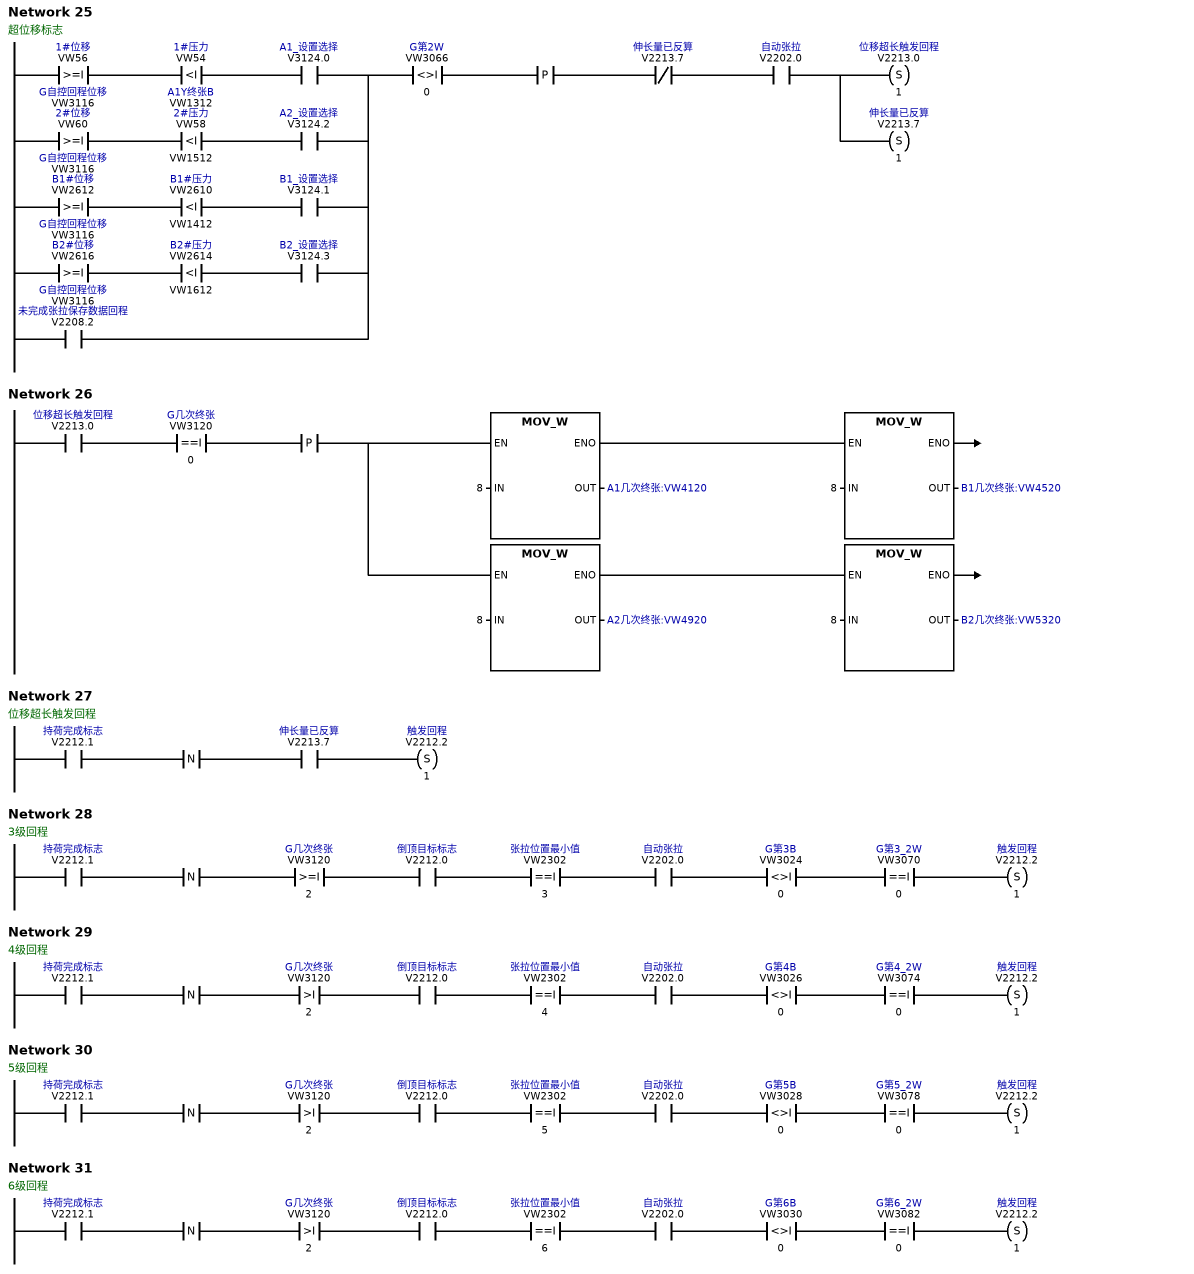
[picture p24: SBR13 networks 25-31]
Network 25
// 超位移标志
LDW>=  1#位移:VW56, G自控回程位移:VW3116
AW<    1#压力:VW54, A1Y终张B:VW1312
A      A1_设置选择:V3124.0
LDW>=  2#位移:VW60, G自控回程位移:VW3116
AW<    2#压力:VW58, VW1512
A      A2_设置选择:V3124.2
OLD
LDW>=  B1#位移:VW2612, G自控回程位移:VW3116
AW<    B1#压力:VW2610, VW1412
A      B1_设置选择:V3124.1
OLD
LDW>=  B2#位移:VW2616, G自控回程位移:VW3116
AW<    B2#压力:VW2614, VW1612
A      B2_设置选择:V3124.3
OLD
O      未完成张拉保存数据回程:V2208.2
AW<>   G第2W:VW3066, 0
EU
AN     伸长量已反算:V2213.7
A      自动张拉:V2202.0
S      位移超长触发回程:V2213.0, 1
S      伸长量已反算:V2213.7, 1
Network 26
LD     位移超长触发回程:V2213.0
AW=    G几次终张:VW3120, 0
EU
LPS
MOVW   8, A1几次终张:VW4120
AENO
MOVW   8, B1几次终张:VW4520
LPP
MOVW   8, A2几次终张:VW4920
AENO
MOVW   8, B2几次终张:VW5320
Network 27
// 位移超长触发回程
LD     持荷完成标志:V2212.1
ED
A      伸长量已反算:V2213.7
S      触发回程:V2212.2, 1
Network 28
// 3级回程
LD     持荷完成标志:V2212.1
ED
AW>=   G几次终张:VW3120, 2
A      倒顶目标标志:V2212.0
AW=    张拉位置最小值:VW2302, 3
A      自动张拉:V2202.0
AW<>   G第3B:VW3024, 0
AW=    G第3_2W:VW3070, 0
S      触发回程:V2212.2, 1
Network 29
// 4级回程
LD     持荷完成标志:V2212.1
ED
AW>    G几次终张:VW3120, 2
A      倒顶目标标志:V2212.0
AW=    张拉位置最小值:VW2302, 4
A      自动张拉:V2202.0
AW<>   G第4B:VW3026, 0
AW=    G第4_2W:VW3074, 0
S      触发回程:V2212.2, 1
Network 30
// 5级回程
LD     持荷完成标志:V2212.1
ED
AW>    G几次终张:VW3120, 2
A      倒顶目标标志:V2212.0
AW=    张拉位置最小值:VW2302, 5
A      自动张拉:V2202.0
AW<>   G第5B:VW3028, 0
AW=    G第5_2W:VW3078, 0
S      触发回程:V2212.2, 1
Network 31
// 6级回程
LD     持荷完成标志:V2212.1
ED
AW>    G几次终张:VW3120, 2
A      倒顶目标标志:V2212.0
AW=    张拉位置最小值:VW2302, 6
A      自动张拉:V2202.0
AW<>   G第6B:VW3030, 0
AW=    G第6_2W:VW3082, 0
S      触发回程:V2212.2, 1
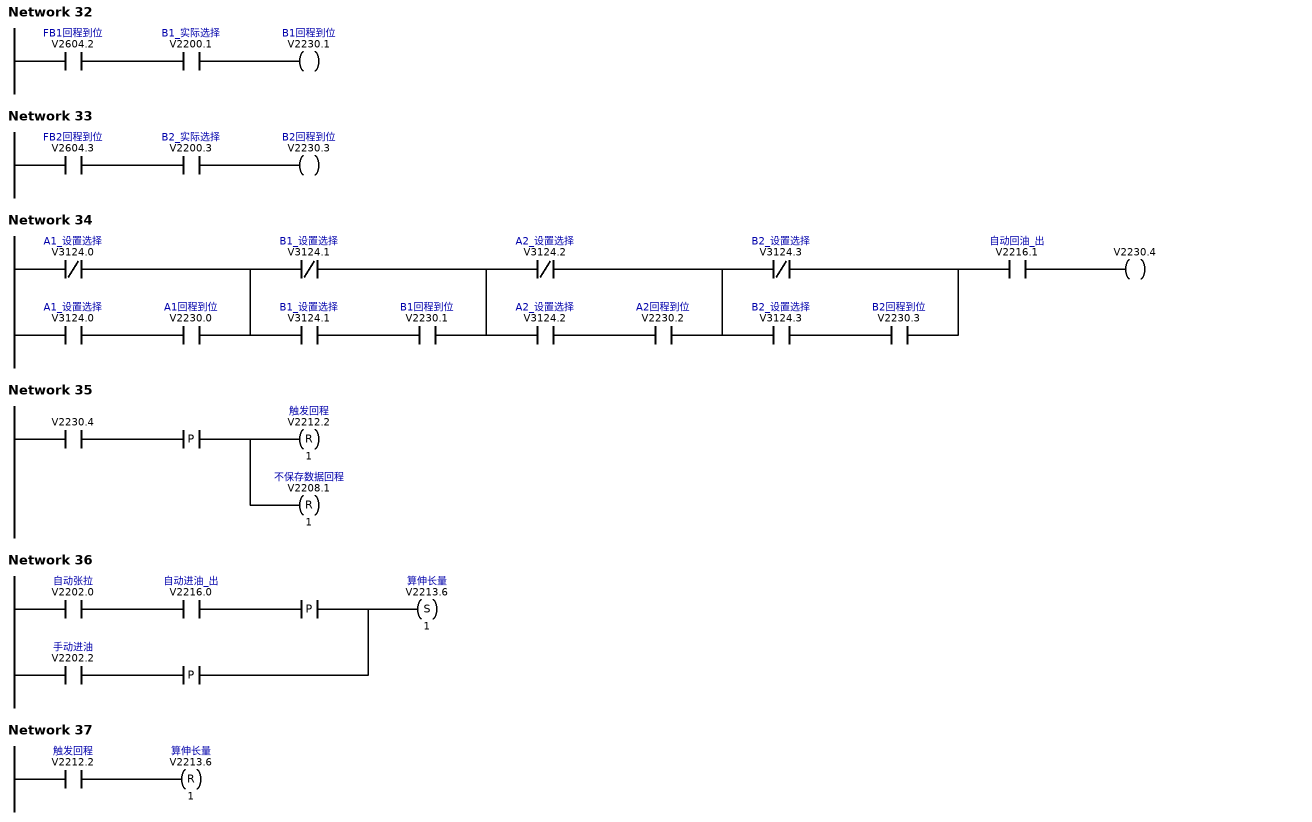
Network 32
LD     FB1回程到位:V2604.2
A      B1_实际选择:V2200.1
=      B1回程到位:V2230.1
Network 33
LD     FB2回程到位:V2604.3
A      B2_实际选择:V2200.3
=      B2回程到位:V2230.3
Network 34
LDN    A1_设置选择:V3124.0
LD     A1_设置选择:V3124.0
A      A1回程到位:V2230.0
OLD
LDN    B1_设置选择:V3124.1
LD     B1_设置选择:V3124.1
A      B1回程到位:V2230.1
OLD
ALD
LDN    A2_设置选择:V3124.2
LD     A2_设置选择:V3124.2
A      A2回程到位:V2230.2
OLD
ALD
LDN    B2_设置选择:V3124.3
LD     B2_设置选择:V3124.3
A      B2回程到位:V2230.3
OLD
ALD
A      自动回油_出:V2216.1
=      V2230.4
Network 35
LD     V2230.4
EU
R      触发回程:V2212.2, 1
R      不保存数据回程:V2208.1, 1
Network 36
LD     自动张拉:V2202.0
A      自动进油_出:V2216.0
EU
LD     手动进油:V2202.2
EU
OLD
S      算伸长量:V2213.6, 1
Network 37
LD     触发回程:V2212.2
R      算伸长量:V2213.6, 1
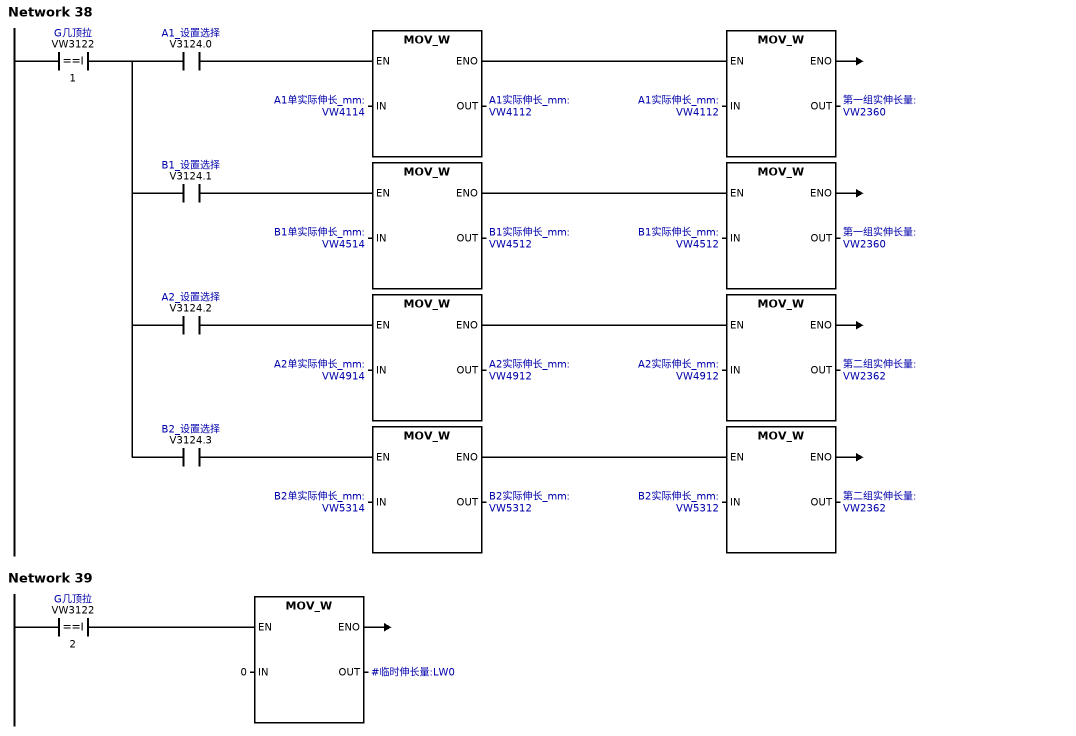
Network 38
LDW=   G几顶拉:VW3122, 1
LPS
A      A1_设置选择:V3124.0
MOVW   A1单实际伸长_mm:VW4114, A1实际伸长_mm:VW4112
AENO
MOVW   A1实际伸长_mm:VW4112, 第一组实伸长量:VW2360
LRD
A      B1_设置选择:V3124.1
MOVW   B1单实际伸长_mm:VW4514, B1实际伸长_mm:VW4512
AENO
MOVW   B1实际伸长_mm:VW4512, 第一组实伸长量:VW2360
LRD
A      A2_设置选择:V3124.2
MOVW   A2单实际伸长_mm:VW4914, A2实际伸长_mm:VW4912
AENO
MOVW   A2实际伸长_mm:VW4912, 第二组实伸长量:VW2362
LPP
A      B2_设置选择:V3124.3
MOVW   B2单实际伸长_mm:VW5314, B2实际伸长_mm:VW5312
AENO
MOVW   B2实际伸长_mm:VW5312, 第二组实伸长量:VW2362
Network 39
LDW=   G几顶拉:VW3122, 2
MOVW   0, #临时伸长量:LW0
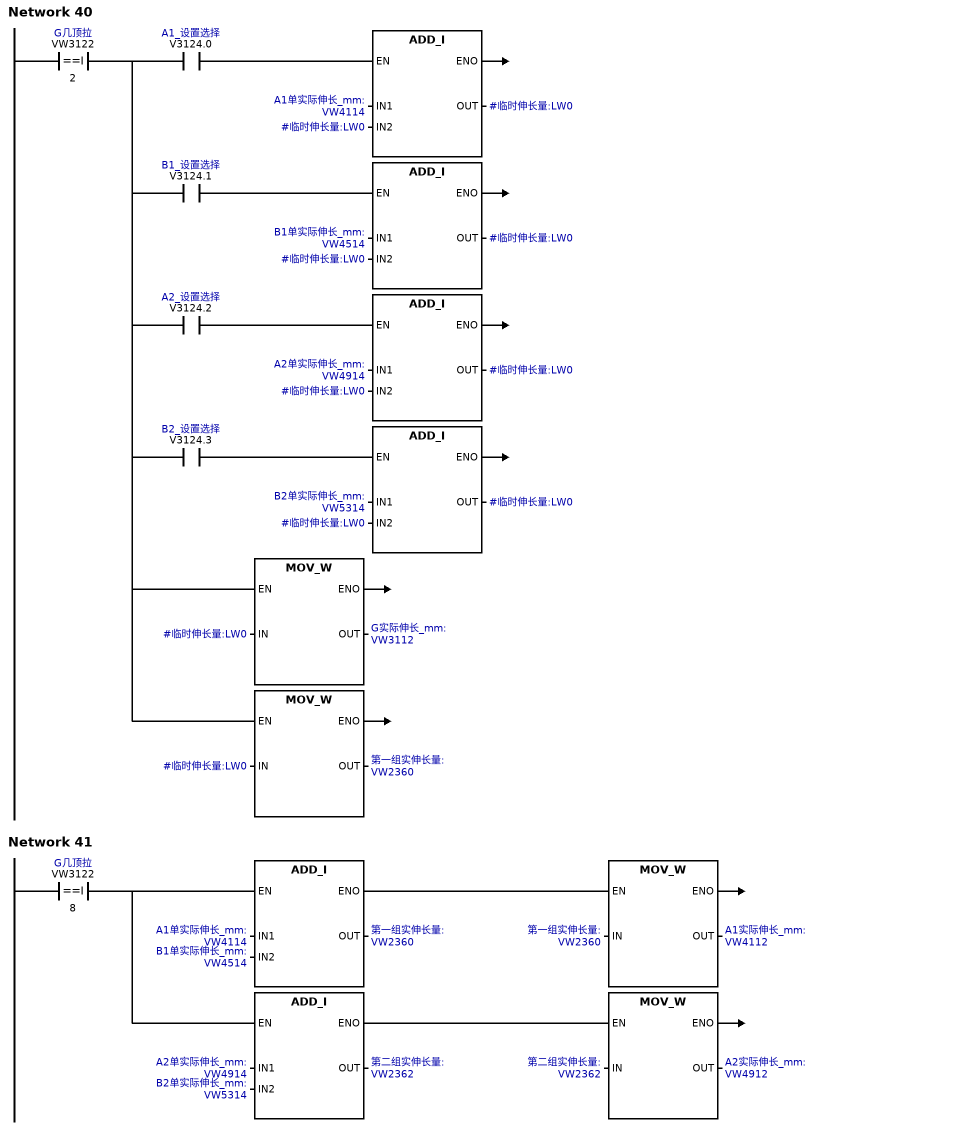
Network 40
LDW=   G几顶拉:VW3122, 2
LPS
A      A1_设置选择:V3124.0
+I     A1单实际伸长_mm:VW4114, #临时伸长量:LW0
LRD
A      B1_设置选择:V3124.1
+I     B1单实际伸长_mm:VW4514, #临时伸长量:LW0
LRD
A      A2_设置选择:V3124.2
+I     A2单实际伸长_mm:VW4914, #临时伸长量:LW0
LRD
A      B2_设置选择:V3124.3
+I     B2单实际伸长_mm:VW5314, #临时伸长量:LW0
LRD
MOVW   #临时伸长量:LW0, G实际伸长_mm:VW3112
LPP
MOVW   #临时伸长量:LW0, 第一组实伸长量:VW2360
Network 41
LDW=   G几顶拉:VW3122, 8
LPS
MOVW   A1单实际伸长_mm:VW4114, 第一组实伸长量:VW2360
AENO
+I     B1单实际伸长_mm:VW4514, 第一组实伸长量:VW2360
AENO
MOVW   第一组实伸长量:VW2360, A1实际伸长_mm:VW4112
LPP
MOVW   A2单实际伸长_mm:VW4914, 第二组实伸长量:VW2362
AENO
+I     B2单实际伸长_mm:VW5314, 第二组实伸长量:VW2362
AENO
MOVW   第二组实伸长量:VW2362, A2实际伸长_mm:VW4912
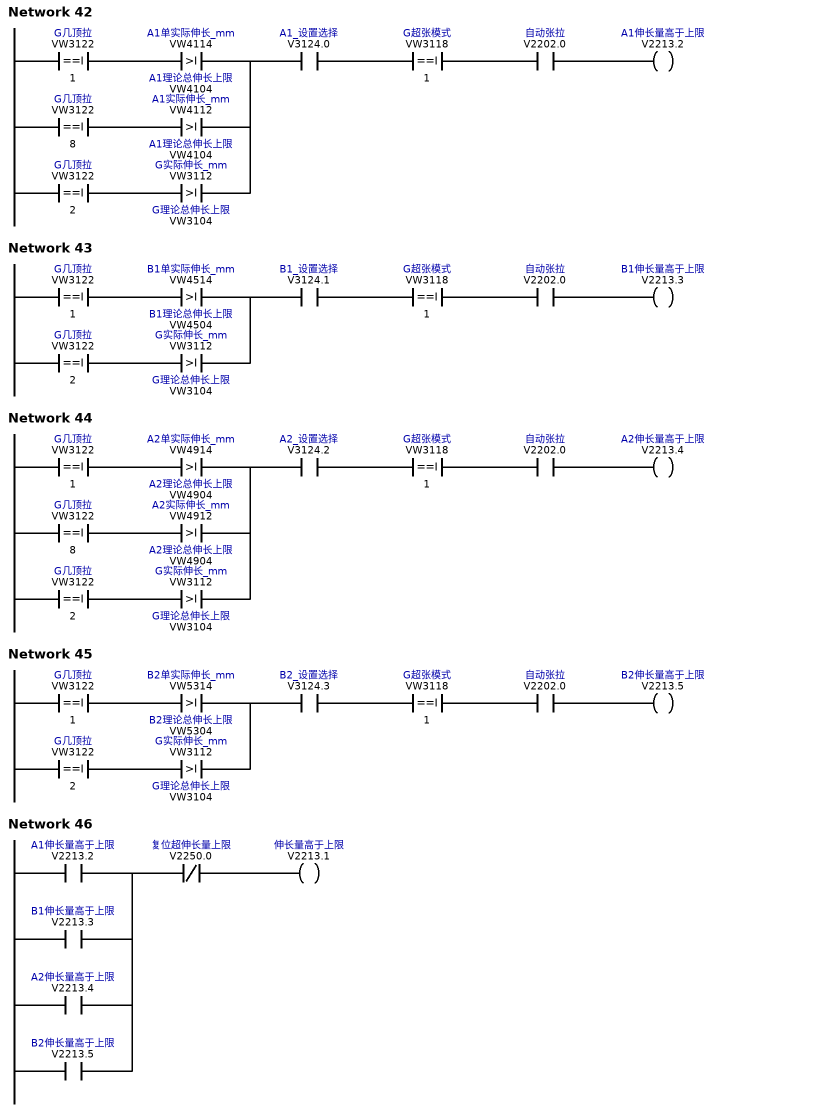
Network 42
LDW=   G几顶拉:VW3122, 1
AW>    A1单实际伸长_mm:VW4114, A1理论总伸长上限:VW4104
LDW=   G几顶拉:VW3122, 8
AW>    A1实际伸长_mm:VW4112, A1理论总伸长上限:VW4104
OLD
LDW=   G几顶拉:VW3122, 2
AW>    G实际伸长_mm:VW3112, G理论总伸长上限:VW3104
OLD
A      A1_设置选择:V3124.0
AW=    G超张模式:VW3118, 1
A      自动张拉:V2202.0
=      A1伸长量高于上限:V2213.2
Network 43
LDW=   G几顶拉:VW3122, 1
AW>    B1单实际伸长_mm:VW4514, B1理论总伸长上限:VW4504
LDW=   G几顶拉:VW3122, 2
AW>    G实际伸长_mm:VW3112, G理论总伸长上限:VW3104
OLD
A      B1_设置选择:V3124.1
AW=    G超张模式:VW3118, 1
A      自动张拉:V2202.0
=      B1伸长量高于上限:V2213.3
Network 44
LDW=   G几顶拉:VW3122, 1
AW>    A2单实际伸长_mm:VW4914, A2理论总伸长上限:VW4904
LDW=   G几顶拉:VW3122, 8
AW>    A2实际伸长_mm:VW4912, A2理论总伸长上限:VW4904
OLD
LDW=   G几顶拉:VW3122, 2
AW>    G实际伸长_mm:VW3112, G理论总伸长上限:VW3104
OLD
A      A2_设置选择:V3124.2
AW=    G超张模式:VW3118, 1
A      自动张拉:V2202.0
=      A2伸长量高于上限:V2213.4
Network 45
LDW=   G几顶拉:VW3122, 1
AW>    B2单实际伸长_mm:VW5314, B2理论总伸长上限:VW5304
LDW=   G几顶拉:VW3122, 2
AW>    G实际伸长_mm:VW3112, G理论总伸长上限:VW3104
OLD
A      B2_设置选择:V3124.3
AW=    G超张模式:VW3118, 1
A      自动张拉:V2202.0
=      B2伸长量高于上限:V2213.5
Network 46
LD     A1伸长量高于上限:V2213.2
O      B1伸长量高于上限:V2213.3
O      A2伸长量高于上限:V2213.4
O      B2伸长量高于上限:V2213.5
AN     复位超伸长量上限:V2250.0
=      伸长量高于上限:V2213.1
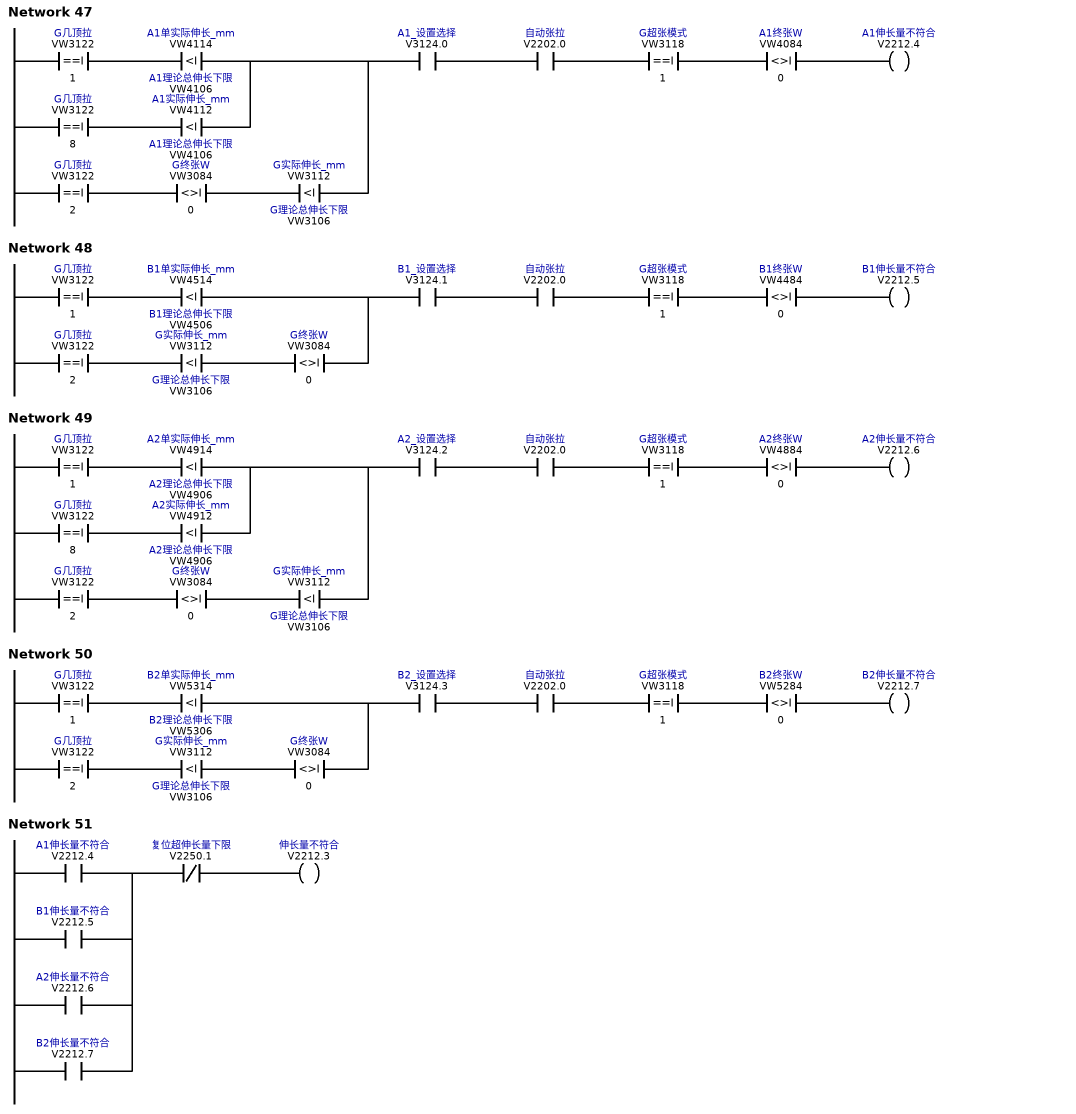
Network 47
LDW=   G几顶拉:VW3122, 1
AW<    A1单实际伸长_mm:VW4114, A1理论总伸长下限:VW4106
LDW=   G几顶拉:VW3122, 8
AW<    A1实际伸长_mm:VW4112, A1理论总伸长下限:VW4106
OLD
LDW=   G几顶拉:VW3122, 2
AW<>   G终张W:VW3084, 0
AW<    G实际伸长_mm:VW3112, G理论总伸长下限:VW3106
OLD
A      A1_设置选择:V3124.0
A      自动张拉:V2202.0
AW=    G超张模式:VW3118, 1
AW<>   A1终张W:VW4084, 0
=      A1伸长量不符合:V2212.4
Network 48
LDW=   G几顶拉:VW3122, 1
AW<    B1单实际伸长_mm:VW4514, B1理论总伸长下限:VW4506
LDW=   G几顶拉:VW3122, 2
AW<    G实际伸长_mm:VW3112, G理论总伸长下限:VW3106
AW<>   G终张W:VW3084, 0
OLD
A      B1_设置选择:V3124.1
A      自动张拉:V2202.0
AW=    G超张模式:VW3118, 1
AW<>   B1终张W:VW4484, 0
=      B1伸长量不符合:V2212.5
Network 49
LDW=   G几顶拉:VW3122, 1
AW<    A2单实际伸长_mm:VW4914, A2理论总伸长下限:VW4906
LDW=   G几顶拉:VW3122, 8
AW<    A2实际伸长_mm:VW4912, A2理论总伸长下限:VW4906
OLD
LDW=   G几顶拉:VW3122, 2
AW<>   G终张W:VW3084, 0
AW<    G实际伸长_mm:VW3112, G理论总伸长下限:VW3106
OLD
A      A2_设置选择:V3124.2
A      自动张拉:V2202.0
AW=    G超张模式:VW3118, 1
AW<>   A2终张W:VW4884, 0
=      A2伸长量不符合:V2212.6
Network 50
LDW=   G几顶拉:VW3122, 1
AW<    B2单实际伸长_mm:VW5314, B2理论总伸长下限:VW5306
LDW=   G几顶拉:VW3122, 2
AW<    G实际伸长_mm:VW3112, G理论总伸长下限:VW3106
AW<>   G终张W:VW3084, 0
OLD
A      B2_设置选择:V3124.3
A      自动张拉:V2202.0
AW=    G超张模式:VW3118, 1
AW<>   B2终张W:VW5284, 0
=      B2伸长量不符合:V2212.7
Network 51
LD     A1伸长量不符合:V2212.4
O      B1伸长量不符合:V2212.5
O      A2伸长量不符合:V2212.6
O      B2伸长量不符合:V2212.7
AN     复位超伸长量下限:V2250.1
=      伸长量不符合:V2212.3
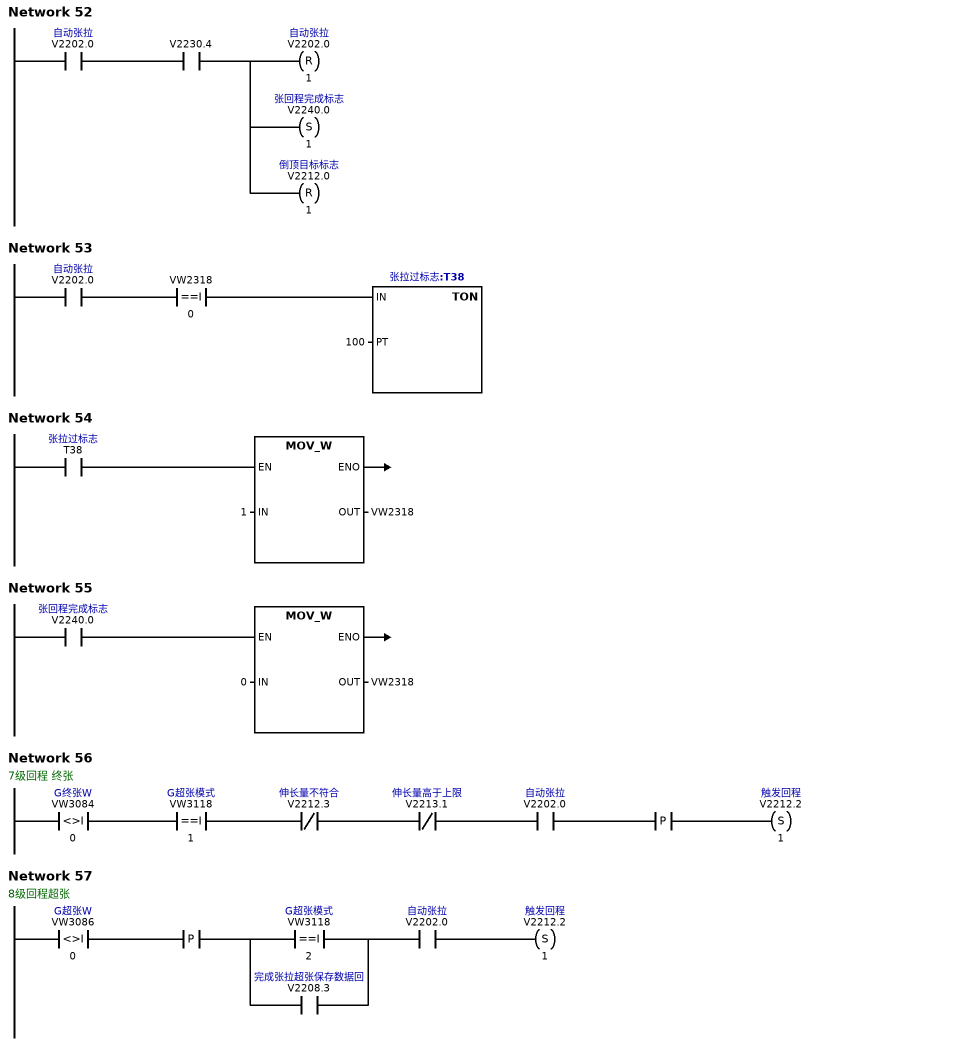
Network 52
LD     自动张拉:V2202.0
A      V2230.4
R      自动张拉:V2202.0, 1
S      张回程完成标志:V2240.0, 1
R      倒顶目标标志:V2212.0, 1
Network 53
LD     自动张拉:V2202.0
AW=    VW2318, 0
TON    张拉过标志:T38, 100
Network 54
LD     张拉过标志:T38
MOVW   1, VW2318
Network 55
LD     张回程完成标志:V2240.0
MOVW   0, VW2318
Network 56
// 7级回程 终张
LDW<>  G终张W:VW3084, 0
AW=    G超张模式:VW3118, 1
AN     伸长量不符合:V2212.3
AN     伸长量高于上限:V2213.1
A      自动张拉:V2202.0
EU
S      触发回程:V2212.2, 1
Network 57
// 8级回程超张
LDW<>  G超张W:VW3086, 0
EU
LDW=   G超张模式:VW3118, 2
O      完成张拉超张保存数据回:V2208.3
ALD
A      自动张拉:V2202.0
S      触发回程:V2212.2, 1
END_SUBROUTINE_BLOCK

SUBROUTINE_BLOCK 自动控制标志:SBR14
TITLE=子程序注释
BEGIN
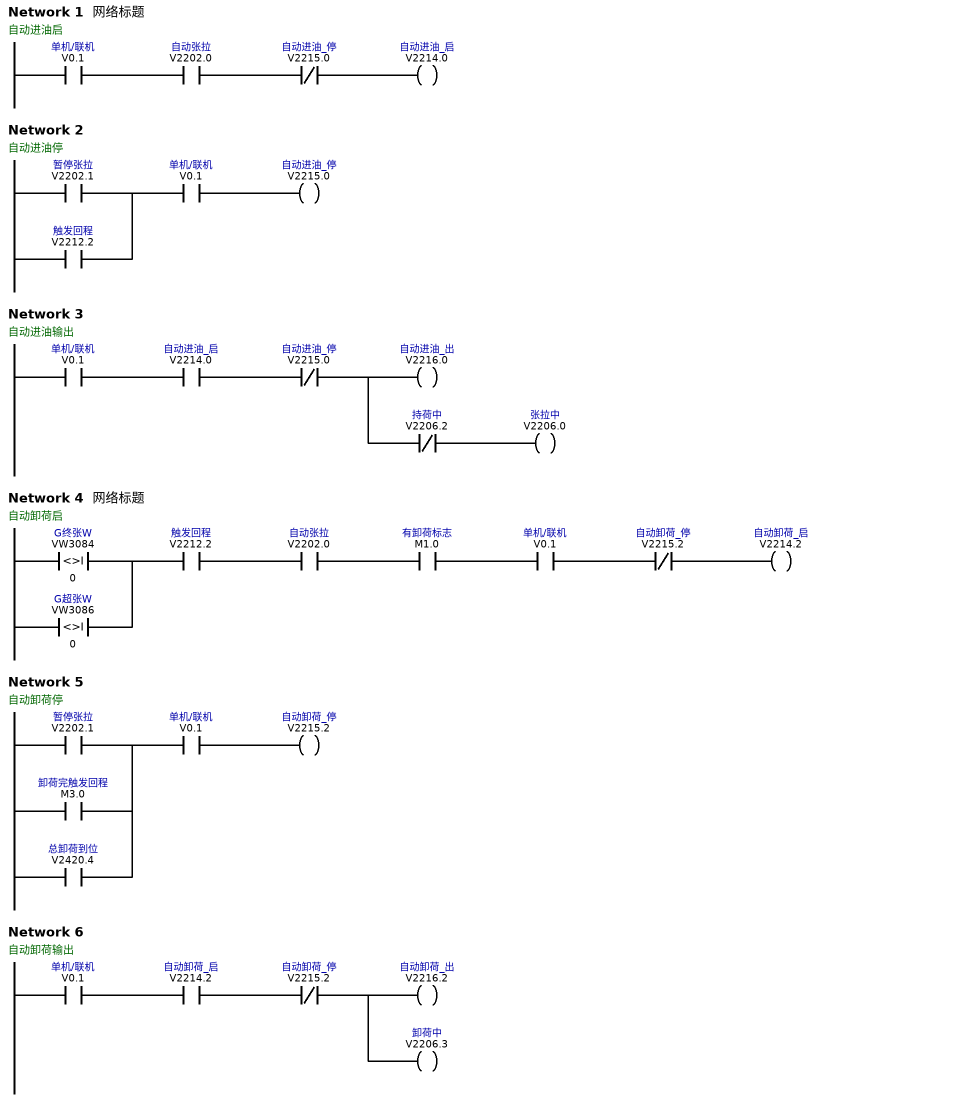
Network 1 // 网络标题
// 自动进油启
LD     单机/联机:V0.1
A      自动张拉:V2202.0
AN     自动进油_停:V2215.0
=      自动进油_启:V2214.0
Network 2
// 自动进油停
LD     暂停张拉:V2202.1
O      触发回程:V2212.2
A      单机/联机:V0.1
=      自动进油_停:V2215.0
Network 3
// 自动进油输出
LD     单机/联机:V0.1
A      自动进油_启:V2214.0
AN     自动进油_停:V2215.0
=      自动进油_出:V2216.0
AN     持荷中:V2206.2
=      张拉中:V2206.0
Network 4 // 网络标题
// 自动卸荷启
LDW<>  G终张W:VW3084, 0
OW<>   G超张W:VW3086, 0
A      触发回程:V2212.2
A      自动张拉:V2202.0
A      有卸荷标志:M1.0
A      单机/联机:V0.1
AN     自动卸荷_停:V2215.2
=      自动卸荷_启:V2214.2
Network 5
// 自动卸荷停
LD     暂停张拉:V2202.1
O      卸荷完触发回程:M3.0
O      总卸荷到位:V2420.4
A      单机/联机:V0.1
=      自动卸荷_停:V2215.2
Network 6
// 自动卸荷输出
LD     单机/联机:V0.1
A      自动卸荷_启:V2214.2
AN     自动卸荷_停:V2215.2
=      自动卸荷_出:V2216.2
=      卸荷中:V2206.3
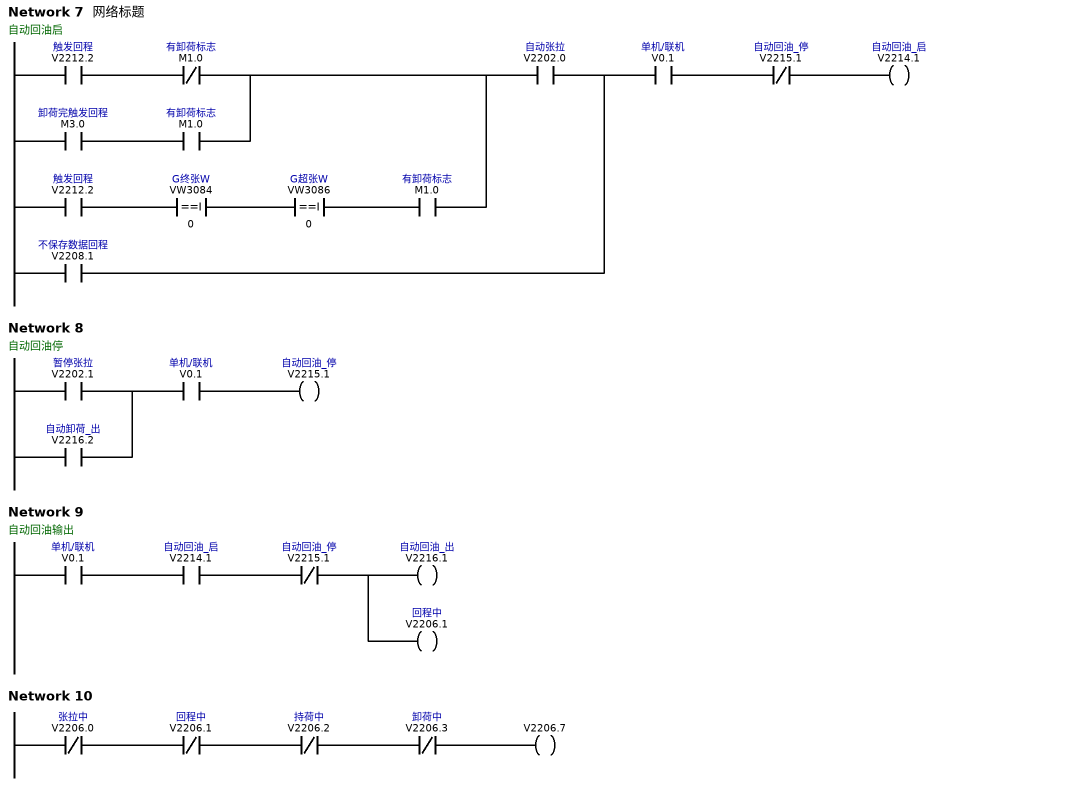
Network 7 // 网络标题
// 自动回油启
LD     触发回程:V2212.2
AN     有卸荷标志:M1.0
LD     卸荷完触发回程:M3.0
A      有卸荷标志:M1.0
OLD
LD     触发回程:V2212.2
AW=    G终张W:VW3084, 0
AW=    G超张W:VW3086, 0
A      有卸荷标志:M1.0
OLD
A      自动张拉:V2202.0
O      不保存数据回程:V2208.1
A      单机/联机:V0.1
AN     自动回油_停:V2215.1
=      自动回油_启:V2214.1
Network 8
// 自动回油停
LD     暂停张拉:V2202.1
O      自动卸荷_出:V2216.2
A      单机/联机:V0.1
=      自动回油_停:V2215.1
Network 9
// 自动回油输出
LD     单机/联机:V0.1
A      自动回油_启:V2214.1
AN     自动回油_停:V2215.1
=      自动回油_出:V2216.1
=      回程中:V2206.1
Network 10
LDN    张拉中:V2206.0
AN     回程中:V2206.1
AN     持荷中:V2206.2
AN     卸荷中:V2206.3
=      V2206.7
END_SUBROUTINE_BLOCK

SUBROUTINE_BLOCK 反算百分比:SBR15
TITLE=子程序注释
VAR_INPUT
当前力:REAL;	// LD0 
总力:REAL;	// LD4 
END_VAR
VAR_OUTPUT
百分比:INT;	// LW8 
END_VAR
VAR
实数百分比:REAL;	// LD10 
END_VAR
BEGIN
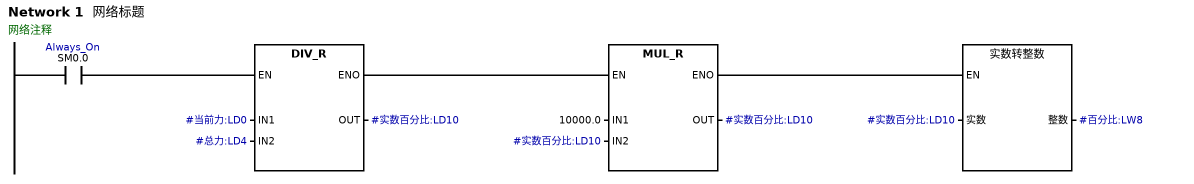
Network 1 // 网络标题
// 网络注释
LD     Always_On:SM0.0
MOVR   #当前力:LD0, #实数百分比:LD10
AENO
/R     #总力:LD4, #实数百分比:LD10
AENO
*R     10000.0, #实数百分比:LD10
AENO
CALL   实数转整数:SBR16, #实数百分比:LD10, #百分比:LW8
END_SUBROUTINE_BLOCK

SUBROUTINE_BLOCK 实数转整数:SBR16
TITLE=子程序注释
VAR_INPUT
实数:REAL;	// LD0 
END_VAR
VAR_OUTPUT
整数:INT;	// LW4 
END_VAR
VAR
双整:DINT;	// LD6 
END_VAR
BEGIN
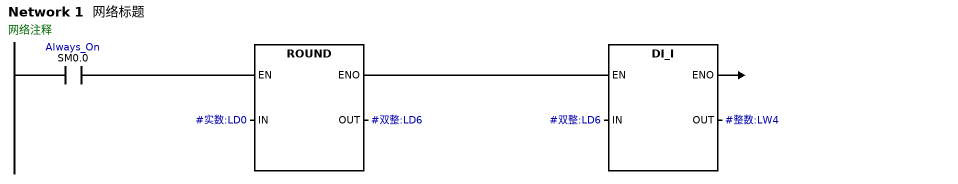
Network 1 // 网络标题
// 网络注释
LD     Always_On:SM0.0
ROUND  #实数:LD0, #双整:LD6
AENO
DTI    #双整:LD6, #整数:LW4
END_SUBROUTINE_BLOCK

SUBROUTINE_BLOCK 计算伸长量:SBR17
TITLE=子程序注释
VAR_INPUT
W1:INT;	// LW0 
W2:INT;	// LW2 
W3_1:INT;	// LW4 
W3_2:INT;	// LW6 
W4_1:INT;	// LW8 
W4_2:INT;	// LW10 
W5_1:INT;	// LW12 
W5_2:INT;	// LW14 
W6_1:INT;	// LW16 
W6_2:INT;	// LW18 
WZZ:INT;	// LW20 
WCZ:INT;	// LW22 
WHS:INT;	// LW24 回缩
当前位移:INT;	// LW26 
WQNSC:INT;	// LW28 千斤顶内伸长量
END_VAR
VAR_OUTPUT
伸长量:INT;	// LW30 
END_VAR
VAR
临时伸长量:INT;	// LW32 
w3差值:INT;	// LW34 
w4差值:INT;	// LW36 
w5差值:INT;	// LW38 
w6差值:INT;	// LW40 
最终值:INT;	// LW42 
初始位移和:INT;	// LW44 
END_VAR
BEGIN
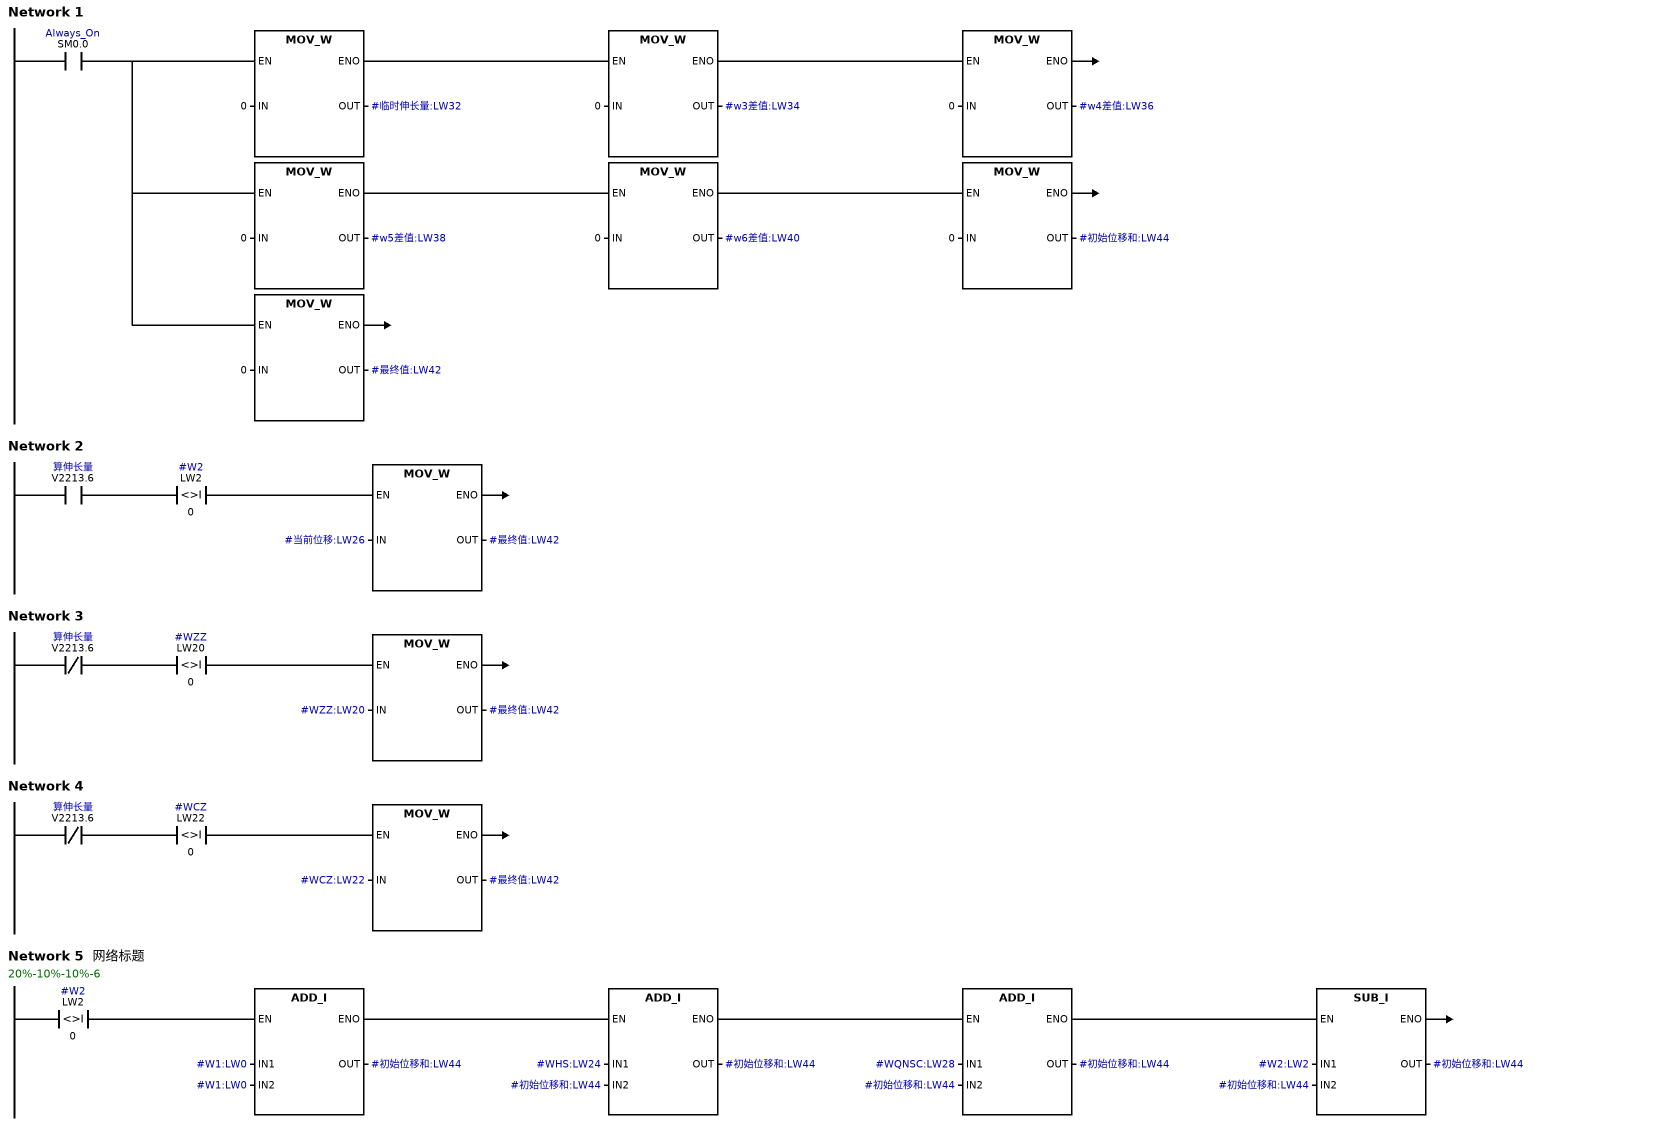
Network 1
LD     Always_On:SM0.0
LPS
MOVW   0, #临时伸长量:LW32
AENO
MOVW   0, #w3差值:LW34
AENO
MOVW   0, #w4差值:LW36
LRD
MOVW   0, #w5差值:LW38
AENO
MOVW   0, #w6差值:LW40
AENO
MOVW   0, #初始位移和:LW44
LPP
MOVW   0, #最终值:LW42
Network 2
LD     算伸长量:V2213.6
AW<>   #W2:LW2, 0
MOVW   #当前位移:LW26, #最终值:LW42
Network 3
LDN    算伸长量:V2213.6
AW<>   #WZZ:LW20, 0
MOVW   #WZZ:LW20, #最终值:LW42
Network 4
LDN    算伸长量:V2213.6
AW<>   #WCZ:LW22, 0
MOVW   #WCZ:LW22, #最终值:LW42
Network 5 // 网络标题
// 20%-10%-10%-6
LDW<>  #W2:LW2, 0
MOVW   #W1:LW0, #初始位移和:LW44
AENO
+I     #W1:LW0, #初始位移和:LW44
AENO
+I     #WHS:LW24, #初始位移和:LW44
AENO
+I     #WQNSC:LW28, #初始位移和:LW44
AENO
INVW   #初始位移和:LW44
INCW   #初始位移和:LW44
+I     #W2:LW2, #初始位移和:LW44
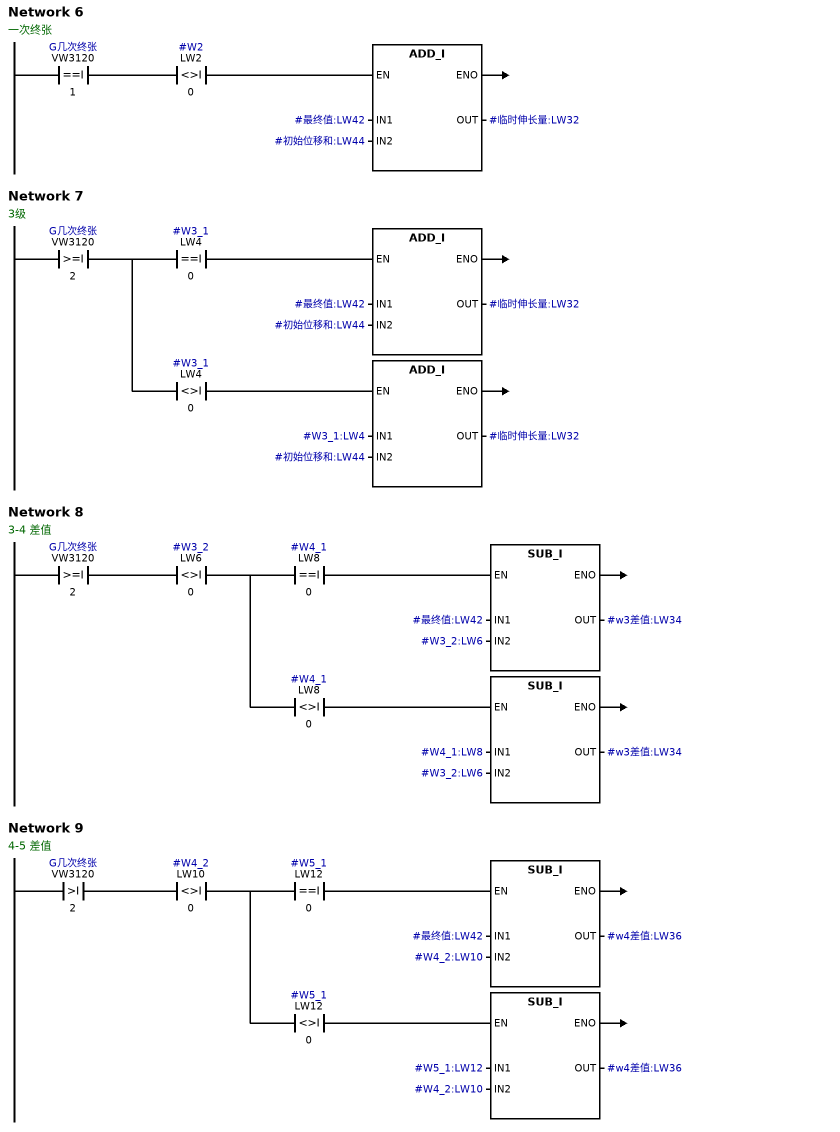
Network 6
// 一次终张
LDW=   G几次终张:VW3120, 1
AW<>   #W2:LW2, 0
MOVW   #最终值:LW42, #临时伸长量:LW32
+I     #初始位移和:LW44, #临时伸长量:LW32
Network 7
// 3级
LDW>=  G几次终张:VW3120, 2
LPS
AW=    #W3_1:LW4, 0
MOVW   #最终值:LW42, #临时伸长量:LW32
+I     #初始位移和:LW44, #临时伸长量:LW32
LPP
AW<>   #W3_1:LW4, 0
MOVW   #W3_1:LW4, #临时伸长量:LW32
+I     #初始位移和:LW44, #临时伸长量:LW32
Network 8
// 3-4 差值
LDW>=  G几次终张:VW3120, 2
AW<>   #W3_2:LW6, 0
LPS
AW=    #W4_1:LW8, 0
MOVW   #最终值:LW42, #w3差值:LW34
-I     #W3_2:LW6, #w3差值:LW34
LPP
AW<>   #W4_1:LW8, 0
MOVW   #W4_1:LW8, #w3差值:LW34
-I     #W3_2:LW6, #w3差值:LW34
Network 9
// 4-5 差值
LDW>   G几次终张:VW3120, 2
AW<>   #W4_2:LW10, 0
LPS
AW=    #W5_1:LW12, 0
MOVW   #最终值:LW42, #w4差值:LW36
-I     #W4_2:LW10, #w4差值:LW36
LPP
AW<>   #W5_1:LW12, 0
MOVW   #W5_1:LW12, #w4差值:LW36
-I     #W4_2:LW10, #w4差值:LW36
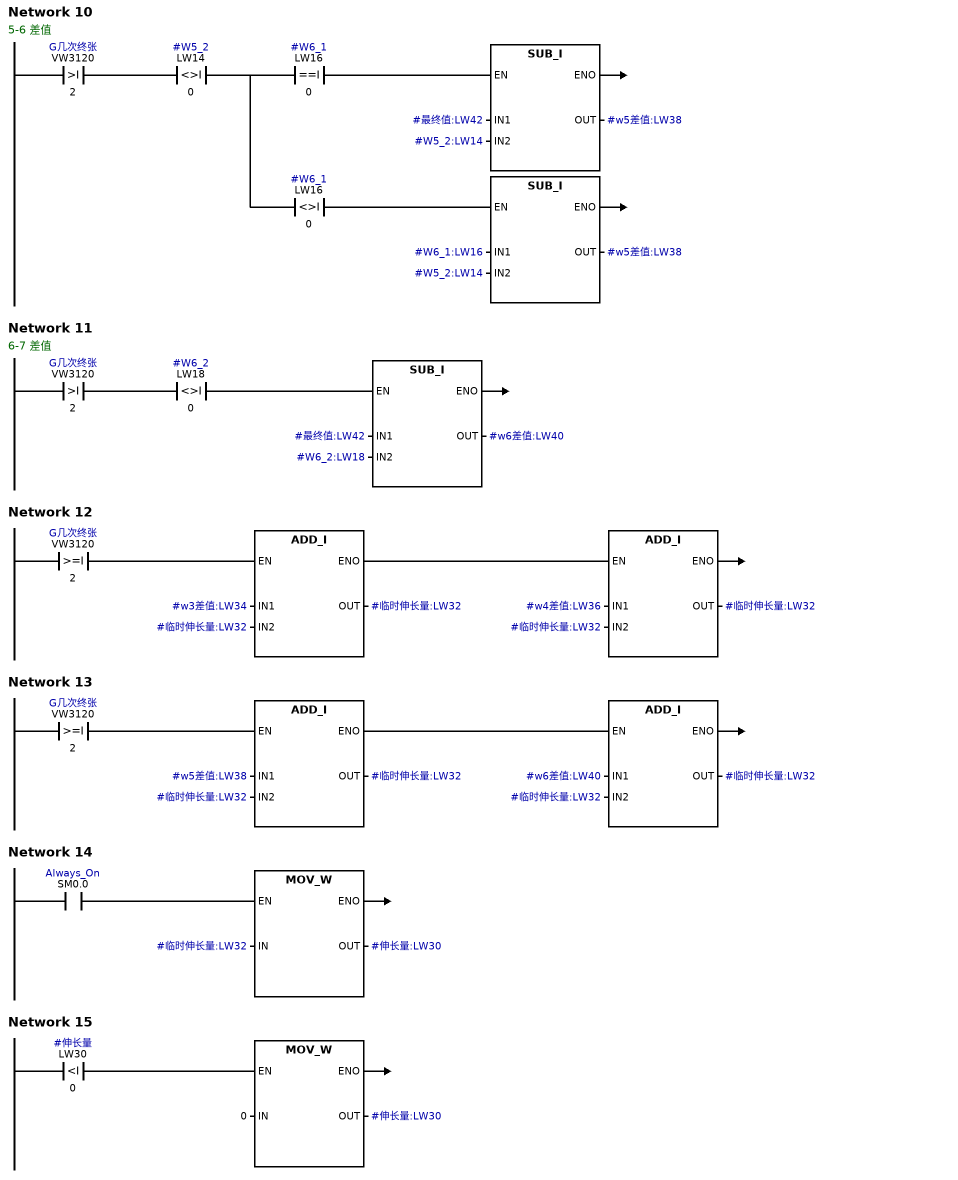
Network 10
// 5-6 差值
LDW>   G几次终张:VW3120, 2
AW<>   #W5_2:LW14, 0
LPS
AW=    #W6_1:LW16, 0
MOVW   #最终值:LW42, #w5差值:LW38
-I     #W5_2:LW14, #w5差值:LW38
LPP
AW<>   #W6_1:LW16, 0
MOVW   #W6_1:LW16, #w5差值:LW38
-I     #W5_2:LW14, #w5差值:LW38
Network 11
// 6-7 差值
LDW>   G几次终张:VW3120, 2
AW<>   #W6_2:LW18, 0
MOVW   #最终值:LW42, #w6差值:LW40
-I     #W6_2:LW18, #w6差值:LW40
Network 12
LDW>=  G几次终张:VW3120, 2
+I     #w3差值:LW34, #临时伸长量:LW32
AENO
+I     #w4差值:LW36, #临时伸长量:LW32
Network 13
LDW>=  G几次终张:VW3120, 2
+I     #w5差值:LW38, #临时伸长量:LW32
AENO
+I     #w6差值:LW40, #临时伸长量:LW32
Network 14
LD     Always_On:SM0.0
MOVW   #临时伸长量:LW32, #伸长量:LW30
Network 15
LDW<   #伸长量:LW30, 0
MOVW   0, #伸长量:LW30
END_SUBROUTINE_BLOCK

SUBROUTINE_BLOCK 主与触摸屏:SBR18
TITLE=子程序注释
VAR
触发记录:BOOL;	// L0.0 
END_VAR
BEGIN
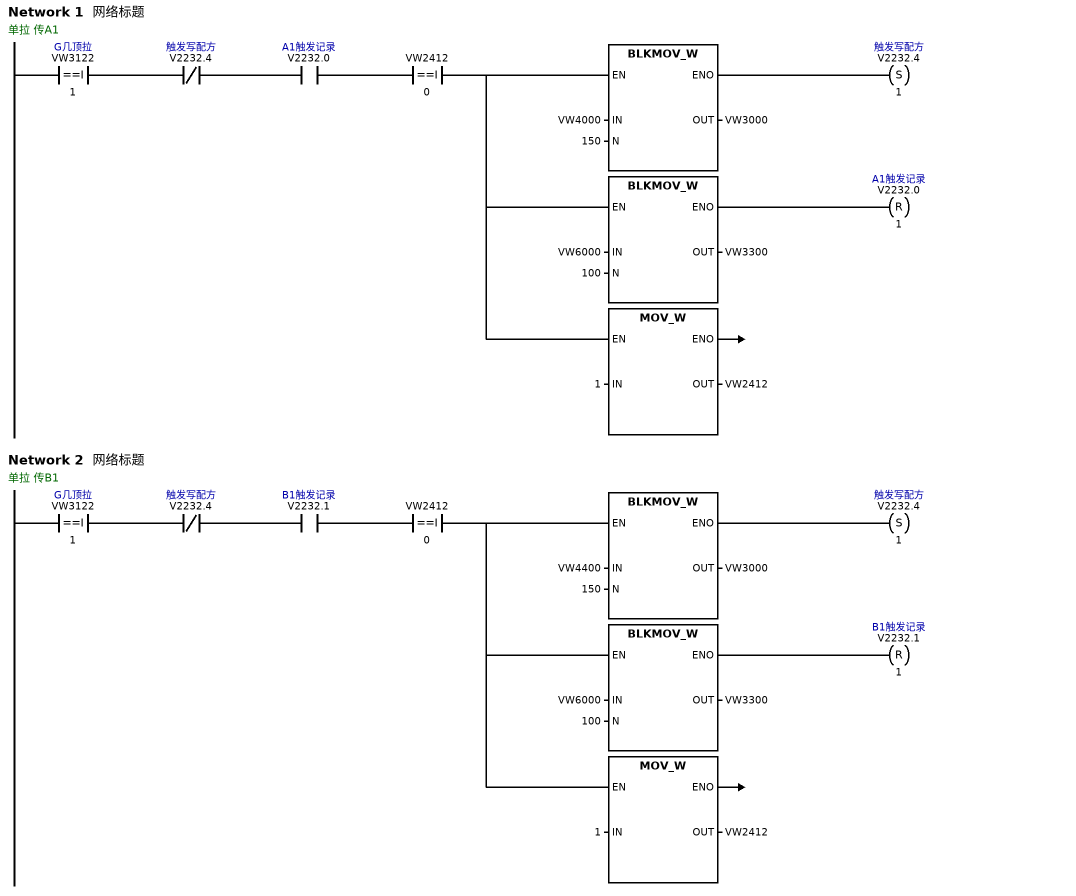
Network 1 // 网络标题
// 单拉 传A1
LDW=   G几顶拉:VW3122, 1
AN     触发写配方:V2232.4
A      A1触发记录:V2232.0
AW=    VW2412, 0
LPS
BMW    VW4000, VW3000, 150
AENO
S      触发写配方:V2232.4, 1
LRD
BMW    VW6000, VW3300, 100
AENO
R      A1触发记录:V2232.0, 1
LPP
MOVW   1, VW2412
Network 2 // 网络标题
// 单拉 传B1
LDW=   G几顶拉:VW3122, 1
AN     触发写配方:V2232.4
A      B1触发记录:V2232.1
AW=    VW2412, 0
LPS
BMW    VW4400, VW3000, 150
AENO
S      触发写配方:V2232.4, 1
LRD
BMW    VW6000, VW3300, 100
AENO
R      B1触发记录:V2232.1, 1
LPP
MOVW   1, VW2412
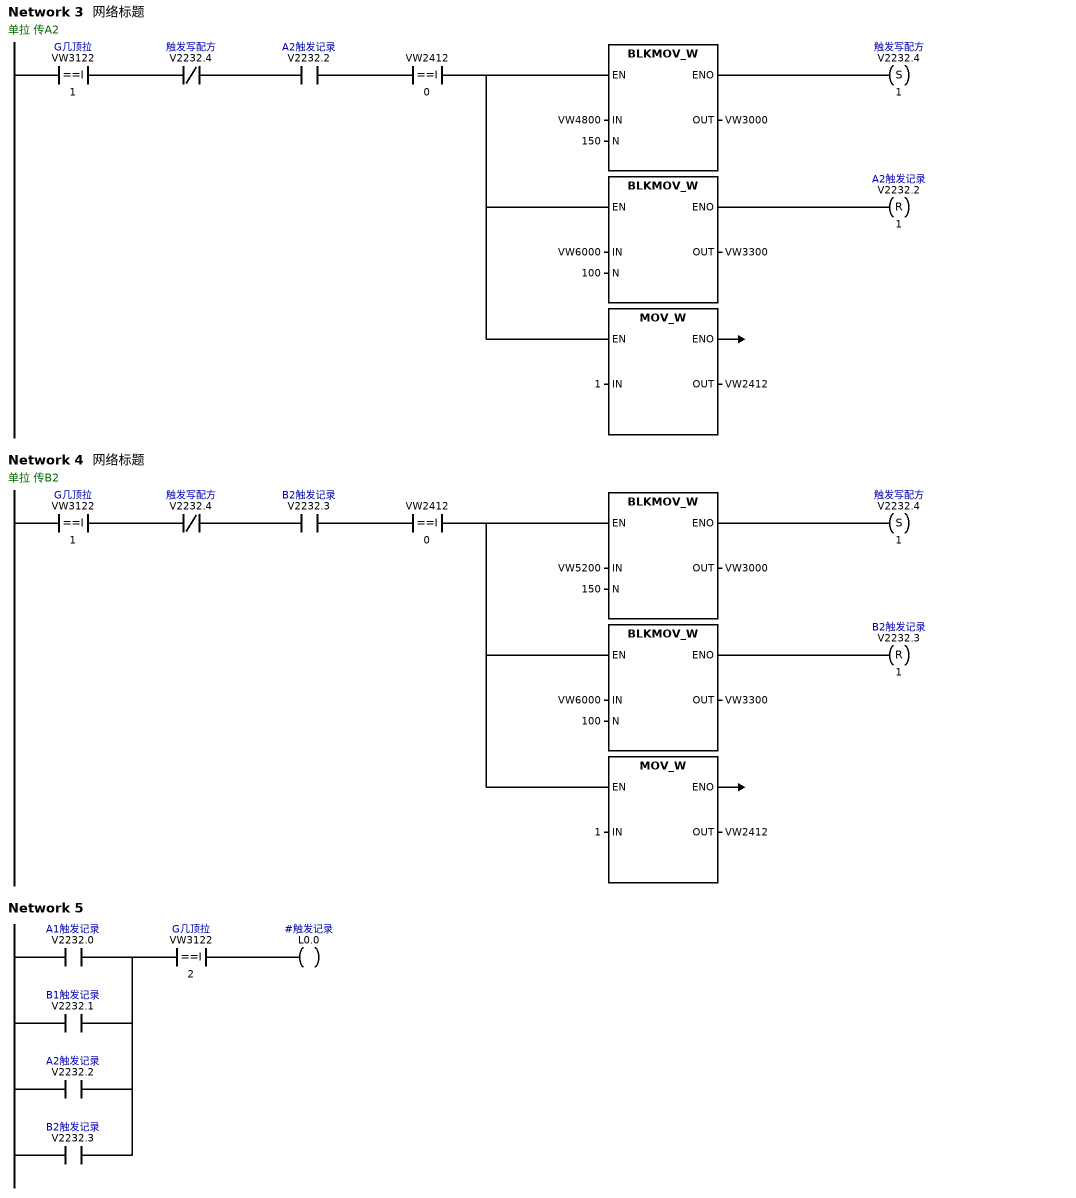
Network 3 // 网络标题
// 单拉 传A2
LDW=   G几顶拉:VW3122, 1
AN     触发写配方:V2232.4
A      A2触发记录:V2232.2
AW=    VW2412, 0
LPS
BMW    VW4800, VW3000, 150
AENO
S      触发写配方:V2232.4, 1
LRD
BMW    VW6000, VW3300, 100
AENO
R      A2触发记录:V2232.2, 1
LPP
MOVW   1, VW2412
Network 4 // 网络标题
// 单拉 传B2
LDW=   G几顶拉:VW3122, 1
AN     触发写配方:V2232.4
A      B2触发记录:V2232.3
AW=    VW2412, 0
LPS
BMW    VW5200, VW3000, 150
AENO
S      触发写配方:V2232.4, 1
LRD
BMW    VW6000, VW3300, 100
AENO
R      B2触发记录:V2232.3, 1
LPP
MOVW   1, VW2412
Network 5
LD     A1触发记录:V2232.0
O      B1触发记录:V2232.1
O      A2触发记录:V2232.2
O      B2触发记录:V2232.3
AW=    G几顶拉:VW3122, 2
=      #触发记录:L0.0
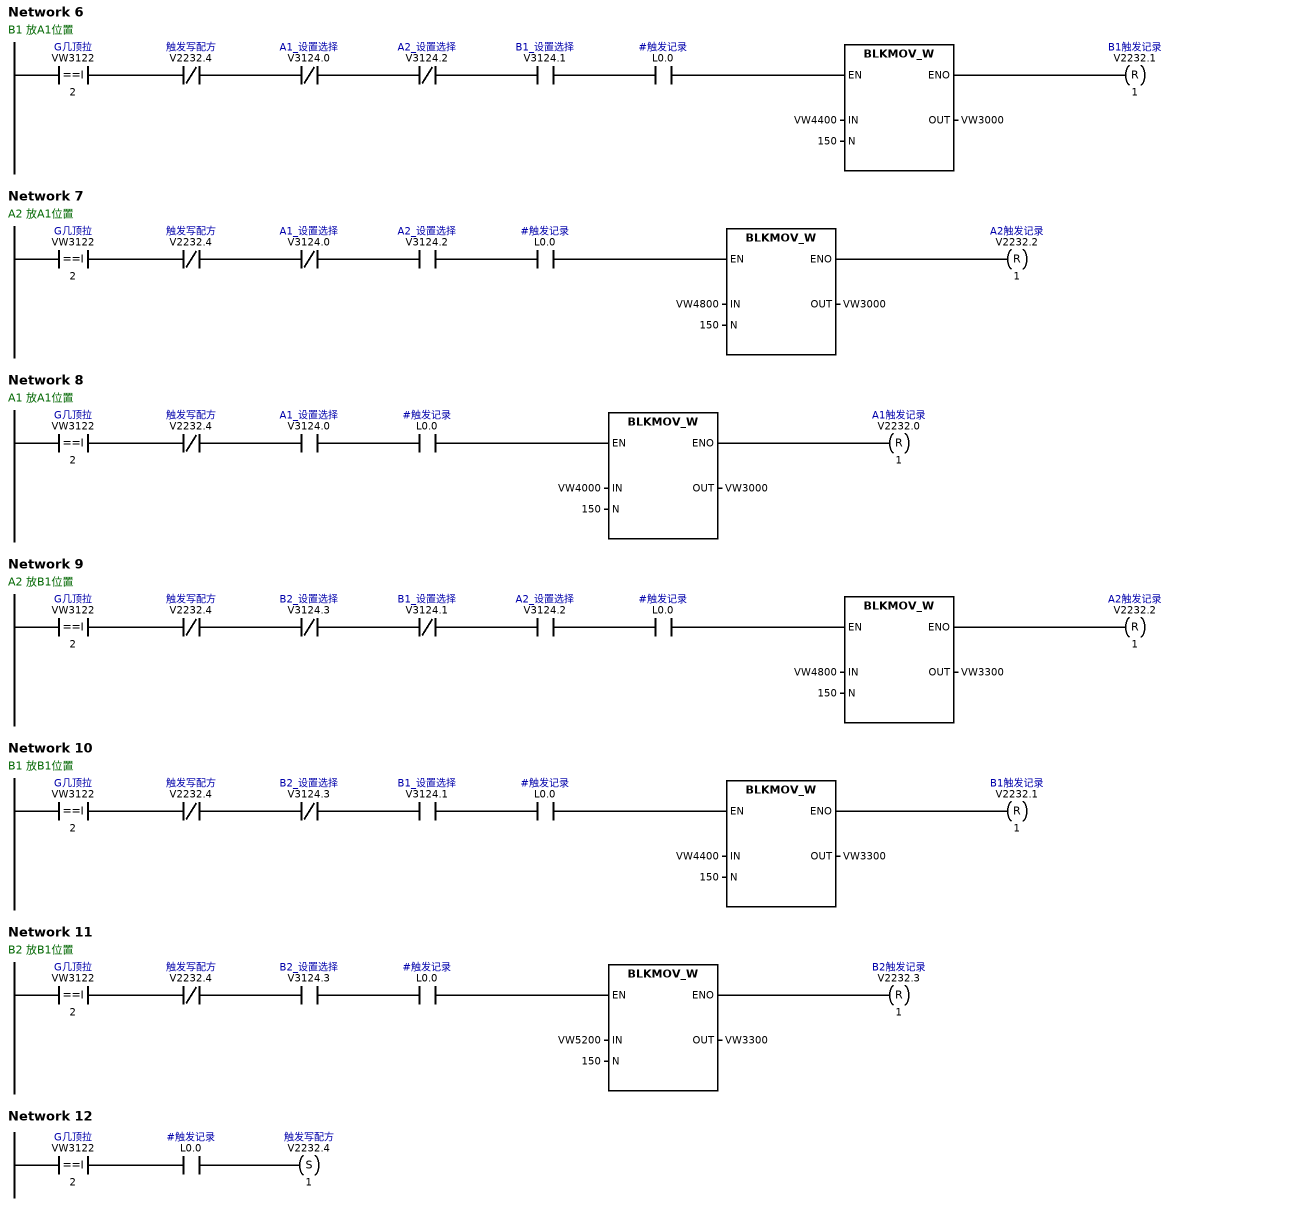
Network 6
// B1 放A1位置
LDW=   G几顶拉:VW3122, 2
AN     触发写配方:V2232.4
AN     A1_设置选择:V3124.0
AN     A2_设置选择:V3124.2
A      B1_设置选择:V3124.1
A      #触发记录:L0.0
BMW    VW4400, VW3000, 150
AENO
R      B1触发记录:V2232.1, 1
Network 7
// A2 放A1位置
LDW=   G几顶拉:VW3122, 2
AN     触发写配方:V2232.4
AN     A1_设置选择:V3124.0
A      A2_设置选择:V3124.2
A      #触发记录:L0.0
BMW    VW4800, VW3000, 150
AENO
R      A2触发记录:V2232.2, 1
Network 8
// A1 放A1位置
LDW=   G几顶拉:VW3122, 2
AN     触发写配方:V2232.4
A      A1_设置选择:V3124.0
A      #触发记录:L0.0
BMW    VW4000, VW3000, 150
AENO
R      A1触发记录:V2232.0, 1
Network 9
// A2 放B1位置
LDW=   G几顶拉:VW3122, 2
AN     触发写配方:V2232.4
AN     B2_设置选择:V3124.3
AN     B1_设置选择:V3124.1
A      A2_设置选择:V3124.2
A      #触发记录:L0.0
BMW    VW4800, VW3300, 150
AENO
R      A2触发记录:V2232.2, 1
Network 10
// B1 放B1位置
LDW=   G几顶拉:VW3122, 2
AN     触发写配方:V2232.4
AN     B2_设置选择:V3124.3
A      B1_设置选择:V3124.1
A      #触发记录:L0.0
BMW    VW4400, VW3300, 150
AENO
R      B1触发记录:V2232.1, 1
Network 11
// B2 放B1位置
LDW=   G几顶拉:VW3122, 2
AN     触发写配方:V2232.4
A      B2_设置选择:V3124.3
A      #触发记录:L0.0
BMW    VW5200, VW3300, 150
AENO
R      B2触发记录:V2232.3, 1
Network 12
LDW=   G几顶拉:VW3122, 2
A      #触发记录:L0.0
S      触发写配方:V2232.4, 1
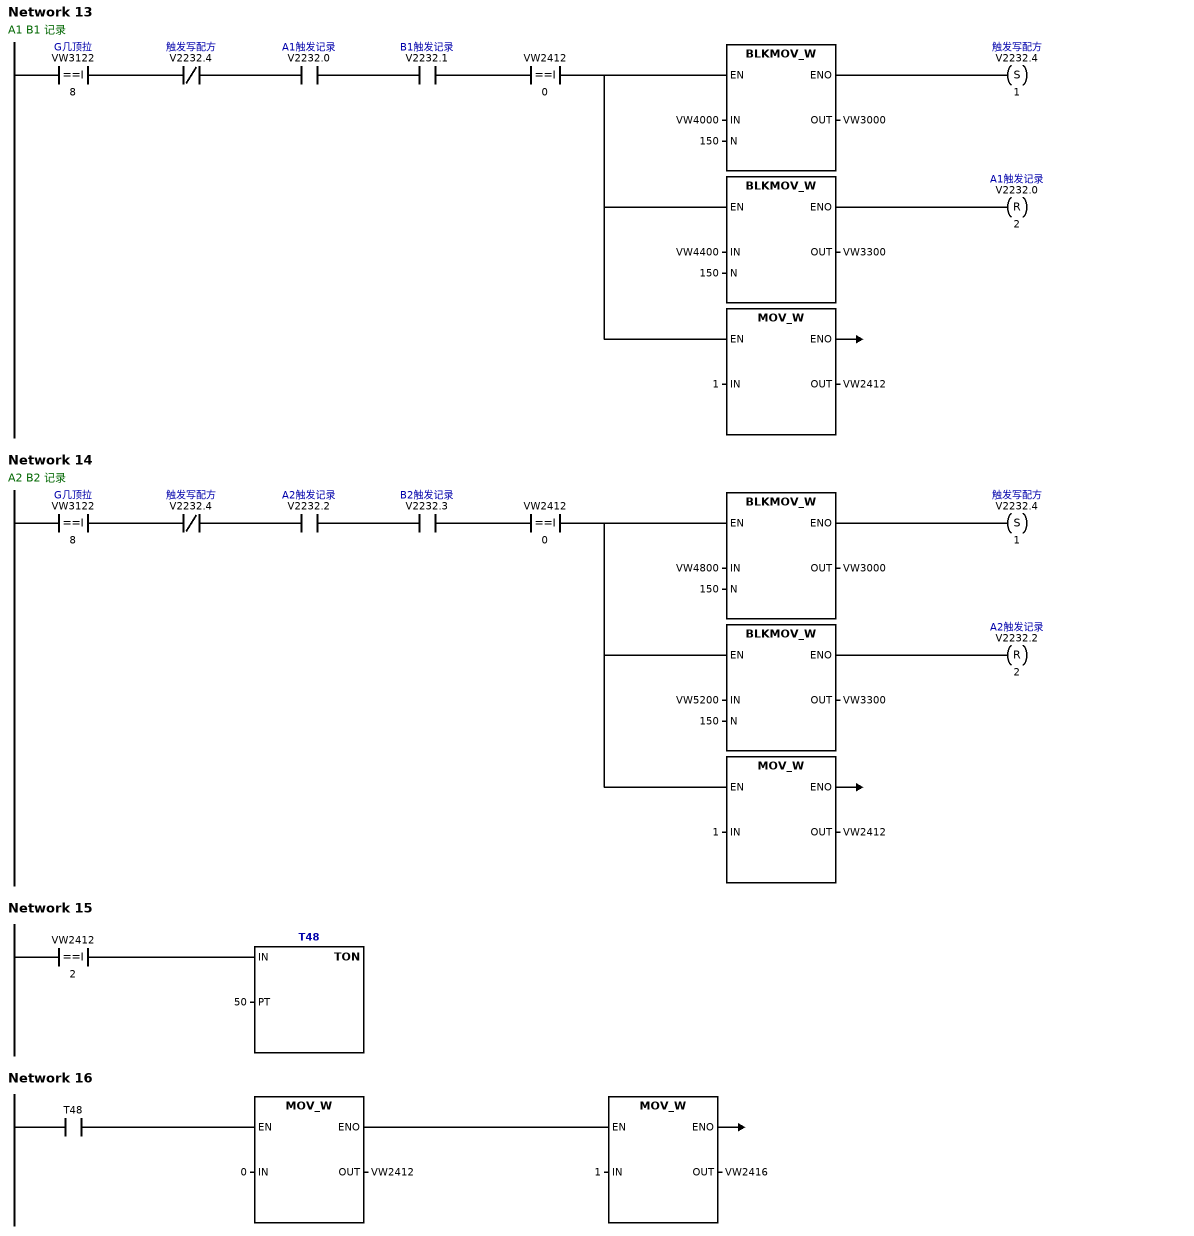
Network 13
// A1 B1 记录
LDW=   G几顶拉:VW3122, 8
AN     触发写配方:V2232.4
A      A1触发记录:V2232.0
A      B1触发记录:V2232.1
AW=    VW2412, 0
LPS
BMW    VW4000, VW3000, 150
AENO
S      触发写配方:V2232.4, 1
LRD
BMW    VW4400, VW3300, 150
AENO
R      A1触发记录:V2232.0, 2
LPP
MOVW   1, VW2412
Network 14
// A2 B2 记录
LDW=   G几顶拉:VW3122, 8
AN     触发写配方:V2232.4
A      A2触发记录:V2232.2
A      B2触发记录:V2232.3
AW=    VW2412, 0
LPS
BMW    VW4800, VW3000, 150
AENO
S      触发写配方:V2232.4, 1
LRD
BMW    VW5200, VW3300, 150
AENO
R      A2触发记录:V2232.2, 2
LPP
MOVW   1, VW2412
Network 15
LDW=   VW2412, 2
TON    T48, 50
Network 16
LD     T48
MOVW   0, VW2412
AENO
MOVW   1, VW2416
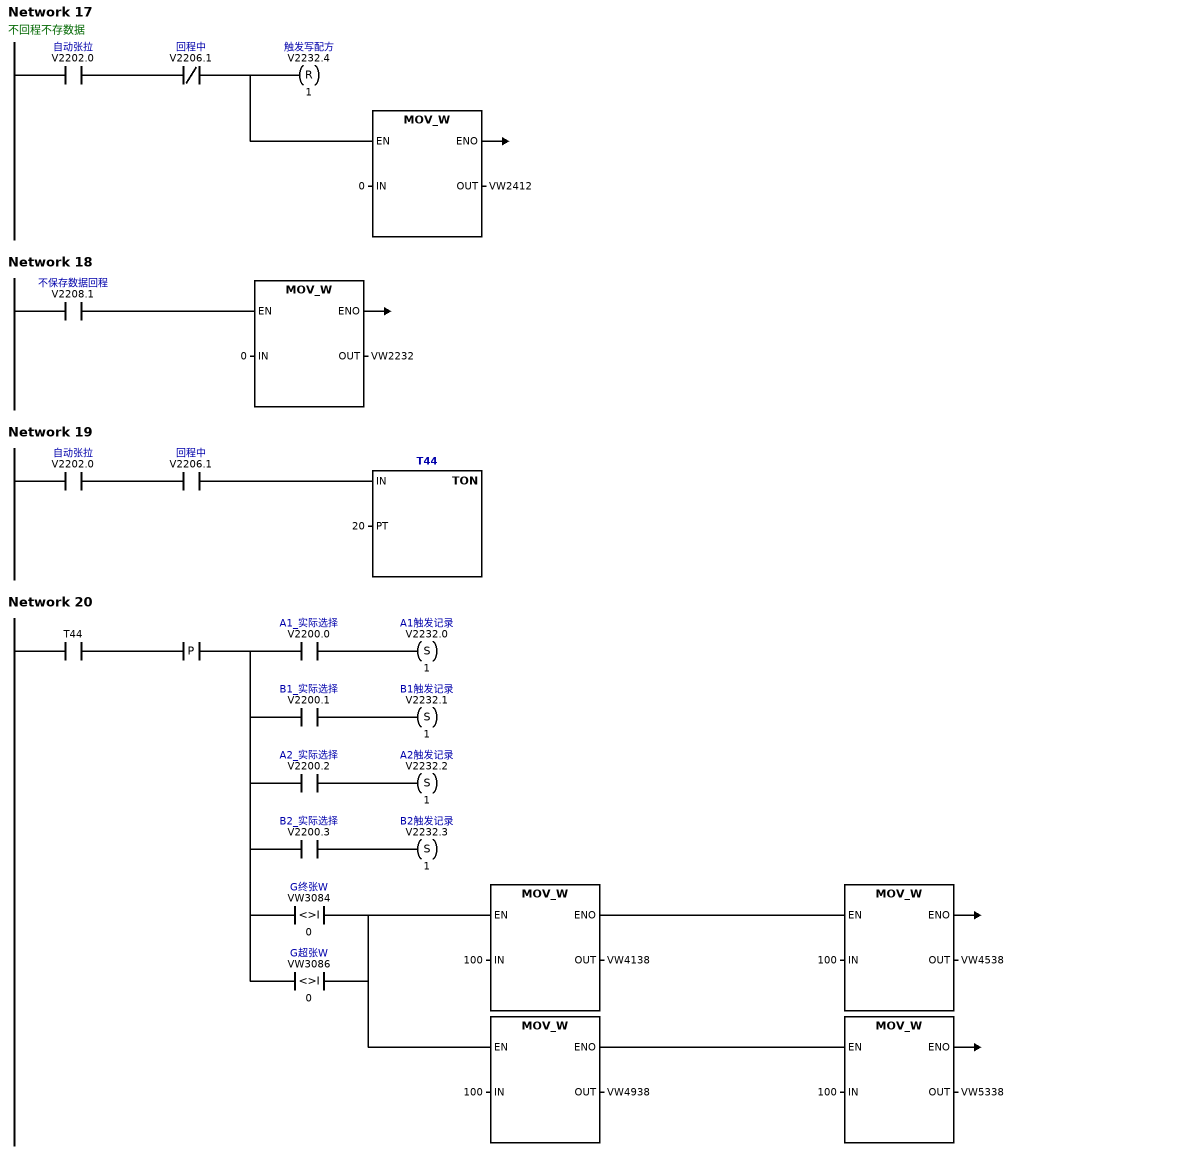
Network 17
// 不回程不存数据
LD     自动张拉:V2202.0
AN     回程中:V2206.1
R      触发写配方:V2232.4, 1
MOVW   0, VW2412
Network 18
LD     不保存数据回程:V2208.1
MOVW   0, VW2232
Network 19
LD     自动张拉:V2202.0
A      回程中:V2206.1
TON    T44, 20
Network 20
LD     T44
EU
LPS
A      A1_实际选择:V2200.0
S      A1触发记录:V2232.0, 1
LRD
A      B1_实际选择:V2200.1
S      B1触发记录:V2232.1, 1
LRD
A      A2_实际选择:V2200.2
S      A2触发记录:V2232.2, 1
LRD
A      B2_实际选择:V2200.3
S      B2触发记录:V2232.3, 1
LPP
LDW<>  G终张W:VW3084, 0
OW<>   G超张W:VW3086, 0
ALD
LPS
MOVW   100, VW4138
AENO
MOVW   100, VW4538
LPP
MOVW   100, VW4938
AENO
MOVW   100, VW5338
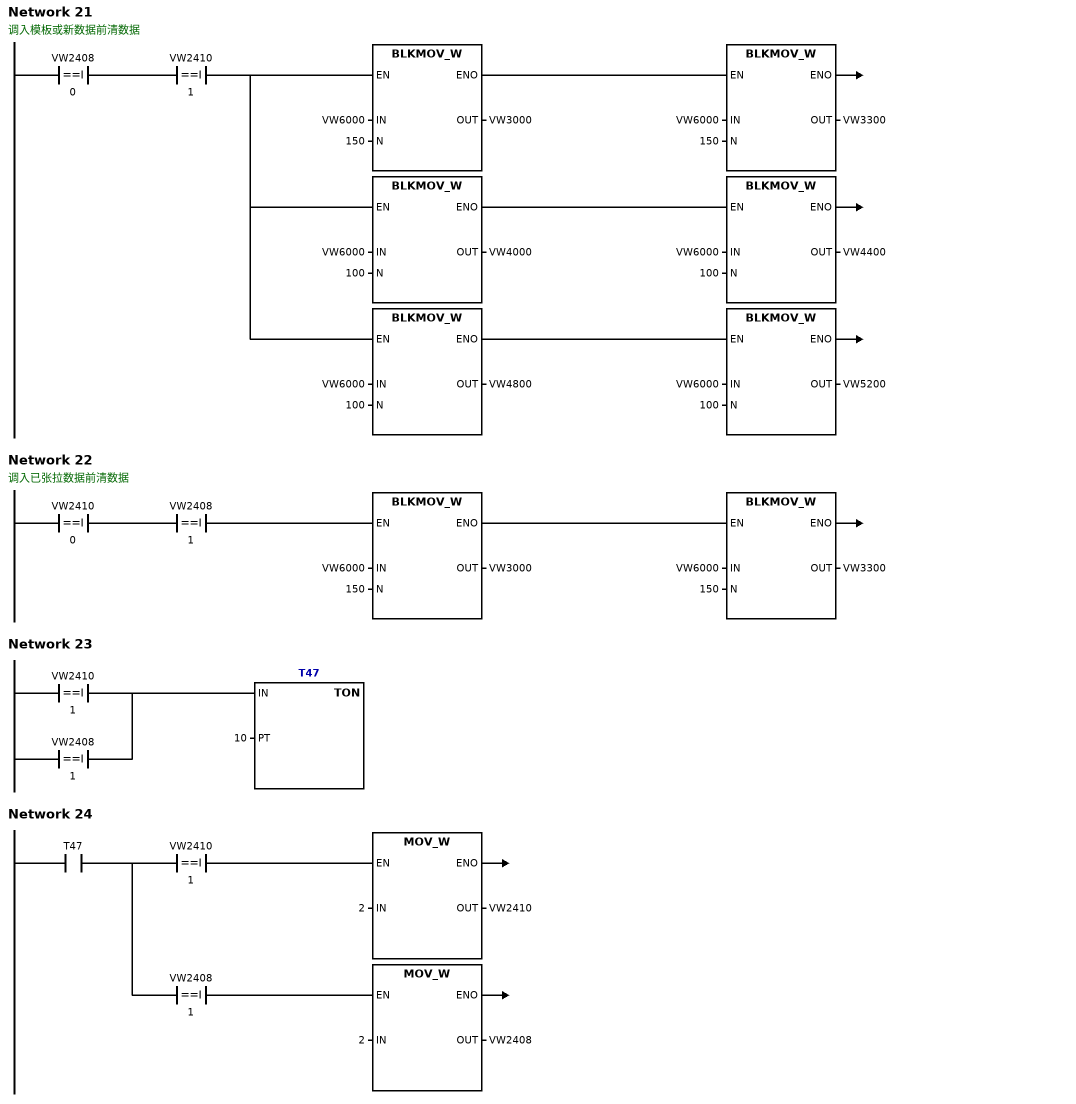
Network 21
// 调入模板或新数据前清数据
LDW=   VW2408, 0
AW=    VW2410, 1
LPS
BMW    VW6000, VW3000, 150
AENO
BMW    VW6000, VW3300, 150
LRD
BMW    VW6000, VW4000, 100
AENO
BMW    VW6000, VW4400, 100
LPP
BMW    VW6000, VW4800, 100
AENO
BMW    VW6000, VW5200, 100
Network 22
// 调入已张拉数据前清数据
LDW=   VW2410, 0
AW=    VW2408, 1
BMW    VW6000, VW3000, 150
AENO
BMW    VW6000, VW3300, 150
Network 23
LDW=   VW2410, 1
OW=    VW2408, 1
TON    T47, 10
Network 24
LD     T47
LPS
AW=    VW2410, 1
MOVW   2, VW2410
LPP
AW=    VW2408, 1
MOVW   2, VW2408
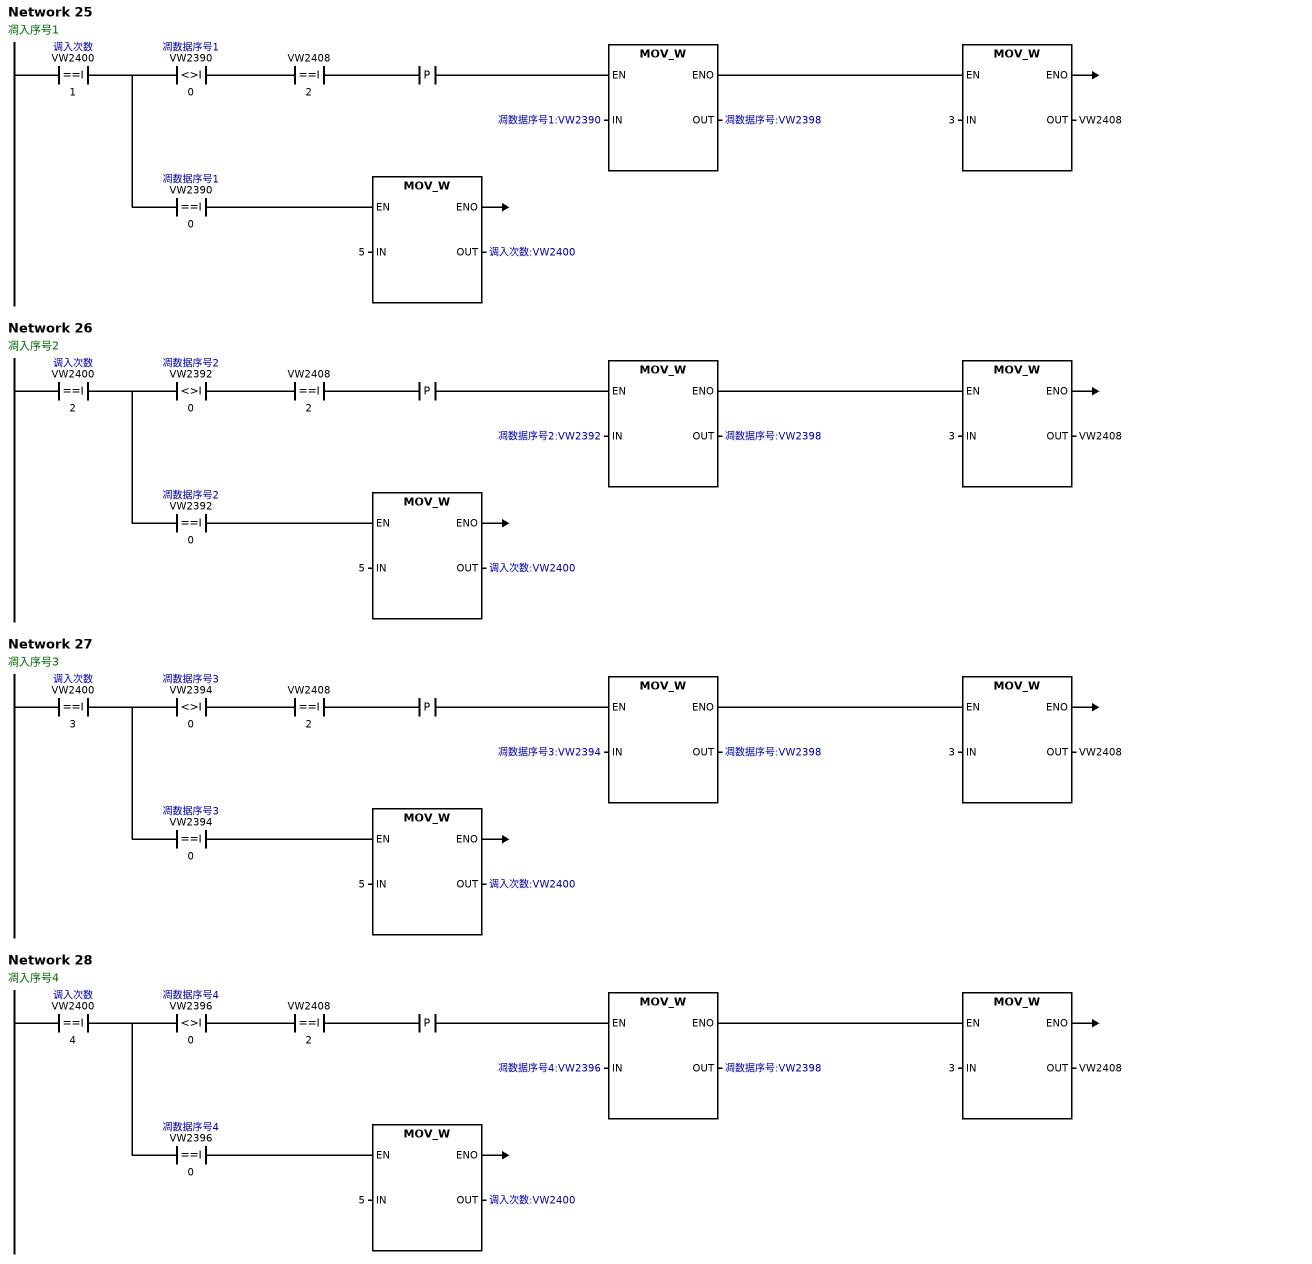
Network 25
// 凋入序号1
LDW=   调入次数:VW2400, 1
LPS
AW<>   凋数据序号1:VW2390, 0
AW=    VW2408, 2
EU
MOVW   凋数据序号1:VW2390, 凋数据序号:VW2398
AENO
MOVW   3, VW2408
LPP
AW=    凋数据序号1:VW2390, 0
MOVW   5, 调入次数:VW2400
Network 26
// 凋入序号2
LDW=   调入次数:VW2400, 2
LPS
AW<>   凋数据序号2:VW2392, 0
AW=    VW2408, 2
EU
MOVW   凋数据序号2:VW2392, 凋数据序号:VW2398
AENO
MOVW   3, VW2408
LPP
AW=    凋数据序号2:VW2392, 0
MOVW   5, 调入次数:VW2400
Network 27
// 凋入序号3
LDW=   调入次数:VW2400, 3
LPS
AW<>   凋数据序号3:VW2394, 0
AW=    VW2408, 2
EU
MOVW   凋数据序号3:VW2394, 凋数据序号:VW2398
AENO
MOVW   3, VW2408
LPP
AW=    凋数据序号3:VW2394, 0
MOVW   5, 调入次数:VW2400
Network 28
// 凋入序号4
LDW=   调入次数:VW2400, 4
LPS
AW<>   凋数据序号4:VW2396, 0
AW=    VW2408, 2
EU
MOVW   凋数据序号4:VW2396, 凋数据序号:VW2398
AENO
MOVW   3, VW2408
LPP
AW=    凋数据序号4:VW2396, 0
MOVW   5, 调入次数:VW2400
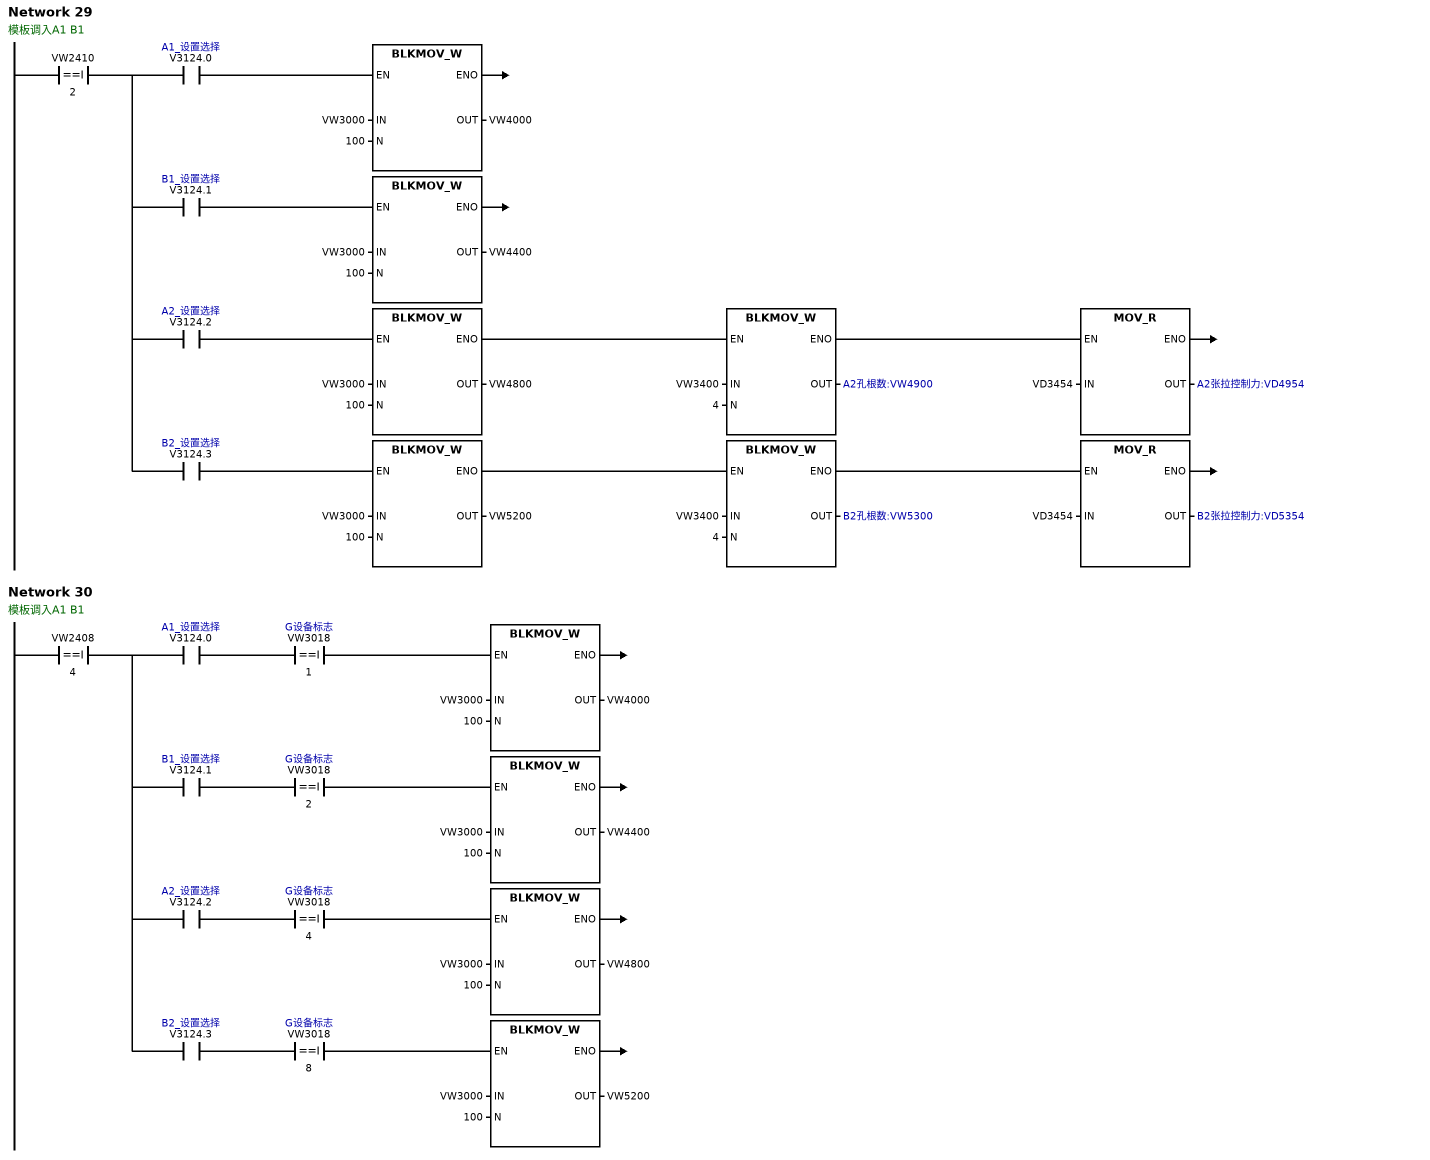
Network 29
// 模板调入A1 B1 
LDW=   VW2410, 2
LPS
A      A1_设置选择:V3124.0
BMW    VW3000, VW4000, 100
LRD
A      B1_设置选择:V3124.1
BMW    VW3000, VW4400, 100
LRD
A      A2_设置选择:V3124.2
BMW    VW3000, VW4800, 100
AENO
BMW    VW3400, A2孔根数:VW4900, 4
AENO
MOVR   VD3454, A2张拉控制力:VD4954
LPP
A      B2_设置选择:V3124.3
BMW    VW3000, VW5200, 100
AENO
BMW    VW3400, B2孔根数:VW5300, 4
AENO
MOVR   VD3454, B2张拉控制力:VD5354
Network 30
// 模板调入A1 B1 
LDW=   VW2408, 4
LPS
A      A1_设置选择:V3124.0
AW=    G设备标志:VW3018, 1
BMW    VW3000, VW4000, 100
LRD
A      B1_设置选择:V3124.1
AW=    G设备标志:VW3018, 2
BMW    VW3000, VW4400, 100
LRD
A      A2_设置选择:V3124.2
AW=    G设备标志:VW3018, 4
BMW    VW3000, VW4800, 100
LPP
A      B2_设置选择:V3124.3
AW=    G设备标志:VW3018, 8
BMW    VW3000, VW5200, 100
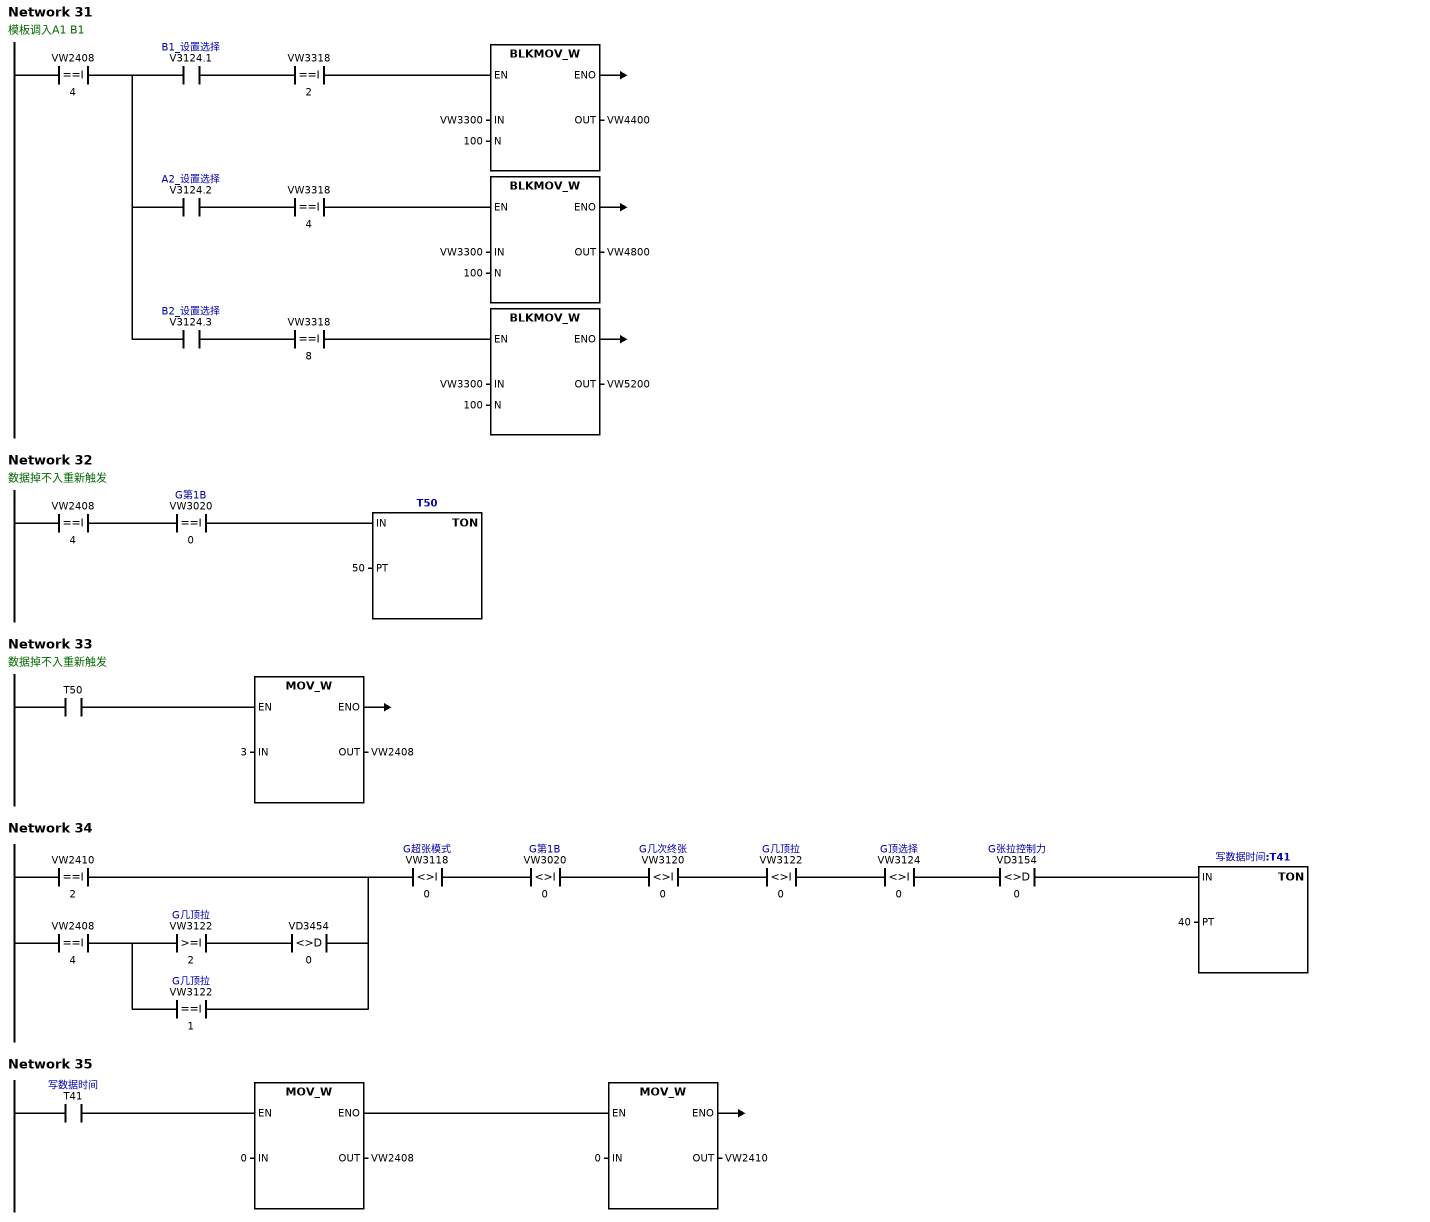
Network 31
// 模板调入A1 B1 
LDW=   VW2408, 4
LPS
A      B1_设置选择:V3124.1
AW=    VW3318, 2
BMW    VW3300, VW4400, 100
LRD
A      A2_设置选择:V3124.2
AW=    VW3318, 4
BMW    VW3300, VW4800, 100
LPP
A      B2_设置选择:V3124.3
AW=    VW3318, 8
BMW    VW3300, VW5200, 100
Network 32
// 数据掉不入重新触发
LDW=   VW2408, 4
AW=    G第1B:VW3020, 0
TON    T50, 50
Network 33
// 数据掉不入重新触发
LD     T50
MOVW   3, VW2408
Network 34
LDW=   VW2410, 2
LDW=   VW2408, 4
LDW>=  G几顶拉:VW3122, 2
AD<>   VD3454, 0
OW=    G几顶拉:VW3122, 1
ALD
OLD
AW<>   G超张模式:VW3118, 0
AW<>   G第1B:VW3020, 0
AW<>   G几次终张:VW3120, 0
AW<>   G几顶拉:VW3122, 0
AW<>   G顶选择:VW3124, 0
AD<>   G张拉控制力:VD3154, 0
TON    写数据时间:T41, 40
Network 35
LD     写数据时间:T41
MOVW   0, VW2408
AENO
MOVW   0, VW2410
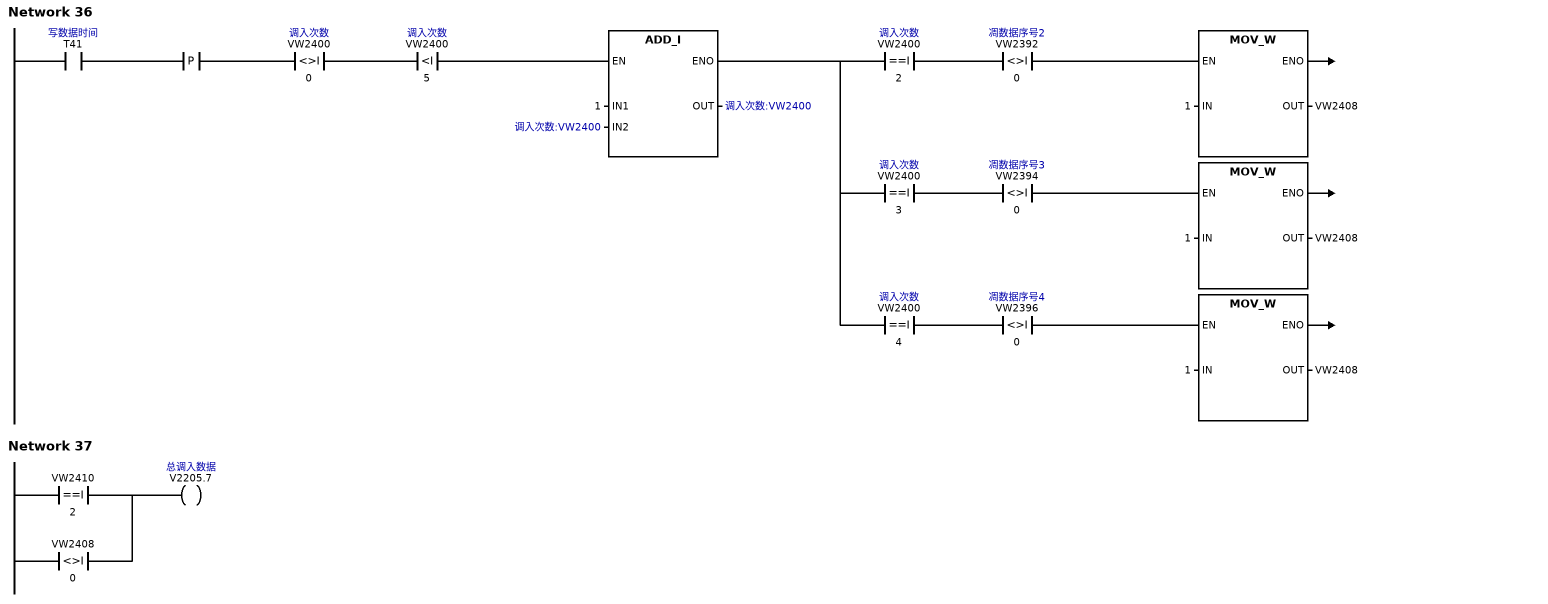
Network 36
LD     写数据时间:T41
EU
AW<>   调入次数:VW2400, 0
AW<    调入次数:VW2400, 5
+I     1, 调入次数:VW2400
AENO
LPS
AW=    调入次数:VW2400, 2
AW<>   凋数据序号2:VW2392, 0
MOVW   1, VW2408
LRD
AW=    调入次数:VW2400, 3
AW<>   凋数据序号3:VW2394, 0
MOVW   1, VW2408
LPP
AW=    调入次数:VW2400, 4
AW<>   凋数据序号4:VW2396, 0
MOVW   1, VW2408
Network 37
LDW=   VW2410, 2
OW<>   VW2408, 0
=      总调入数据:V2205.7
